(* Logix 5000 project; controller test vendor 1 type 14 code 151 rev 32.13; software revision 32.02; part 2 of 4 *)

        [600].Status := 2, [601].Status := 2, [602].Status := 2, [603].Status := 2, [604].Status := 2, [605].Status := 2, [606].Status := 2, [607].Status := 2, [608].Status := 2, [609].Status := 2, [610].Status := 2, [611].Status := 2, [612].Status := 2, [613].Status := 2, [614].Status := 2, [615].Status := 2, [616].Status := 2, [617].Status := 2, [618].Status := 2, [619].Status := 2, [620].Status := 2, [621].Status := 2, [622].Status := 2, [623].Status := 2, [624].Status := 2, [625].Status := 2, [626].Status := 2, [627].Status := 2, [628].Status := 2, [629].Status := 2, [630].Status := 2, [631].Status := 2, [632].Status := 2, [633].Status := 2, [634].Status := 2, [635].Status := 2, [636].Status := 2, [637].Status := 2, [638].Status := 2, [639].Status := 2, [640].Status := 2, [641].Status := 2, [642].Status := 2, [643].Status := 2, [644].Status := 2, [645].Status := 2, [646].Status := 2, [647].Status := 2, [648].Status := 2, [649].Status := 2, [650].Status := 2, [651].Status := 2, [652].Status := 2, [653].Status := 2, [654].Status := 2, [655].Status := 2, [656].Status := 2, [657].Status := 2, [658].Status := 2, [659].Status := 2,
        [660].Status := 2, [661].Status := 2, [662].Status := 2, [663].Status := 2, [664].Status := 2, [665].Status := 2, [666].Status := 2, [667].Status := 2, [668].Status := 2, [669].Status := 2, [670].Status := 2, [671].Status := 2, [672].Status := 2, [673].Status := 2, [674].Status := 2, [675].Status := 2, [676].Status := 2, [677].Status := 2, [678].Status := 2, [679].Status := 2, [680].Status := 2, [681].Status := 2, [682].Status := 2, [683].Status := 2, [684].Status := 2, [685].Status := 2, [686].Status := 2, [687].Status := 2, [688].Status := 2, [689].Status := 2, [690].Status := 2, [691].Status := 2, [692].Status := 2, [693].Status := 2, [694].Status := 2, [695].Status := 2, [696].Status := 2, [697].Status := 2, [698].Status := 2, [699].Status := 2, [700].Status := 2, [701].Status := 2, [702].Status := 2, [703].Status := 2, [704].Status := 2, [705].Status := 2, [706].Status := 2, [707].Status := 2, [708].Status := 2, [709].Status := 2, [710].Status := 2, [711].Status := 2, [712].Status := 2, [713].Status := 2, [714].Status := 2, [715].Status := 2, [716].Status := 2, [717].Status := 2, [718].Status := 2, [719].Status := 2,
        [720].Status := 2, [721].Status := 2, [722].Status := 2, [723].Status := 2, [724].Status := 2, [725].Status := 2, [726].Status := 2, [727].Status := 2, [728].Status := 2, [729].Status := 2, [730].Status := 2, [731].Status := 2, [732].Status := 2, [733].Status := 2, [734].Status := 2, [735].Status := 2, [736].Status := 2, [737].Status := 2, [738].Status := 2, [739].Status := 2, [740].Status := 2, [741].Status := 2, [742].Status := 2, [743].Status := 2, [744].Status := 2, [745].Status := 2, [746].Status := 2, [747].Status := 2, [748].Status := 2, [749].Status := 2, [750].Status := 2, [751].Status := 2, [752].Status := 2, [753].Status := 2, [754].Status := 2, [755].Status := 2, [756].Status := 2, [757].Status := 2, [758].Status := 2, [759].Status := 2, [760].Status := 2, [761].Status := 2, [762].Status := 2, [763].Status := 2, [764].Status := 2, [765].Status := 2, [766].Status := 2, [767].Status := 2, [768].Status := 2, [769].Status := 2, [770].Status := 2, [771].Status := 2, [772].Status := 2, [773].Status := 2, [774].Status := 2, [775].Status := 2, [776].Status := 2, [777].Status := 2, [778].Status := 2, [779].Status := 2,
        [780].Status := 2, [781].Status := 2, [782].Status := 2, [783].Status := 2, [784].Status := 2, [785].Status := 2, [786].Status := 2, [787].Status := 2, [788].Status := 2, [789].Status := 2, [790].Status := 2, [791].Status := 2, [792].Status := 2, [793].Status := 2, [794].Status := 2, [795].Status := 2, [796].Status := 2, [797].Status := 2, [798].Status := 2, [799].Status := 2, [800].Status := 2, [801].Status := 2, [802].Status := 2, [803].Status := 2, [804].Status := 2, [805].Status := 2, [806].Status := 2, [807].Status := 2, [808].Status := 2, [809].Status := 2, [810].Status := 2, [811].Status := 2, [812].Status := 2, [813].Status := 2, [814].Status := 2, [815].Status := 2, [816].Status := 2, [817].Status := 2, [818].Status := 2, [819].Status := 2, [820].Status := 2, [821].Status := 2, [822].Status := 2, [823].Status := 2, [824].Status := 2, [825].Status := 2, [826].Status := 2, [827].Status := 2, [828].Status := 2, [829].Status := 2, [830].Status := 2, [831].Status := 2, [832].Status := 2, [833].Status := 2, [834].Status := 2, [835].Status := 2, [836].Status := 2, [837].Status := 2, [838].Status := 2, [839].Status := 2,
        [840].Status := 2, [841].Status := 2, [842].Status := 2, [843].Status := 2, [844].Status := 2, [845].Status := 2, [846].Status := 2, [847].Status := 2, [848].Status := 2, [849].Status := 2, [850].Status := 2, [851].Status := 2, [852].Status := 2, [853].Status := 2, [854].Status := 2, [855].Status := 2, [856].Status := 2, [857].Status := 2, [858].Status := 2, [859].Status := 2, [860].Status := 2, [861].Status := 2, [862].Status := 2, [863].Status := 2, [864].Status := 2, [865].Status := 2, [866].Status := 2, [867].Status := 2, [868].Status := 2, [869].Status := 2, [870].Status := 2, [871].Status := 2, [872].Status := 2, [873].Status := 2, [874].Status := 2, [875].Status := 2, [876].Status := 2, [877].Status := 2, [878].Status := 2, [879].Status := 2, [880].Status := 2, [881].Status := 2, [882].Status := 2, [883].Status := 2, [884].Status := 2, [885].Status := 2, [886].Status := 2, [887].Status := 2, [888].Status := 2, [889].Status := 2, [890].Status := 2, [891].Status := 2, [892].Status := 2, [893].Status := 2, [894].Status := 2, [895].Status := 2, [896].Status := 2, [897].Status := 2, [898].Status := 2, [899].Status := 2,
        [900].Status := 2, [901].Status := 2, [902].Status := 2, [903].Status := 2, [904].Status := 2, [905].Status := 2, [906].Status := 2, [907].Status := 2, [908].Status := 2, [909].Status := 2, [910].Status := 2, [911].Status := 2, [912].Status := 2, [913].Status := 2, [914].Status := 2, [915].Status := 2, [916].Status := 2, [917].Status := 2, [918].Status := 2, [919].Status := 2, [920].Status := 2, [921].Status := 2, [922].Status := 2, [923].Status := 2, [924].Status := 2, [925].Status := 2, [926].Status := 2, [927].Status := 2, [928].Status := 2, [929].Status := 2, [930].Status := 2, [931].Status := 2, [932].Status := 2, [933].Status := 2, [934].Status := 2, [935].Status := 2, [936].Status := 2, [937].Status := 2, [938].Status := 2, [939].Status := 2, [940].Status := 2, [941].Status := 2, [942].Status := 2, [943].Status := 2, [944].Status := 2, [945].Status := 2, [946].Status := 2, [947].Status := 2, [948].Status := 2, [949].Status := 2, [950].Status := 2, [951].Status := 2, [952].Status := 2, [953].Status := 2, [954].Status := 2, [955].Status := 2, [956].Status := 2, [957].Status := 2, [958].Status := 2, [959].Status := 2,
        [960].Status := 2, [961].Status := 2, [962].Status := 2, [963].Status := 2, [964].Status := 2, [965].Status := 2, [966].Status := 2, [967].Status := 2, [968].Status := 2, [969].Status := 2, [970].Status := 2, [971].Status := 2, [972].Status := 2, [973].Status := 2, [974].Status := 2, [975].Status := 2, [976].Status := 2, [977].Status := 2, [978].Status := 2, [979].Status := 2, [980].Status := 2, [981].Status := 2, [982].Status := 2, [983].Status := 2, [984].Status := 2, [985].Status := 2, [986].Status := 2, [987].Status := 2, [988].Status := 2, [989].Status := 2, [990].Status := 2, [991].Status := 2, [992].Status := 2, [993].Status := 2, [994].Status := 2, [995].Status := 2, [996].Status := 2, [997].Status := 2, [998].Status := 2, [999].Status := 2, [1000].Status := 2, [1001].Status := 2, [1002].Status := 2);
   AlarmPressureHigh : REAL;
   AnalogFlowAirHAlarm : ALIAS FOR Local:2:I.Ch1HAlarm;
   AnalogFlowAirLAlarm : ALIAS FOR Local:2:I.Ch1LAlarm;
   AnalogFlowO2HAlarm : ALIAS FOR Local:2:I.Ch0HAlarm;
   AnalogFlowO2LAlarm : ALIAS FOR Local:2:I.Ch0LAlarm;
   AnalogInputFlow : ALIAS FOR Local:2:I.Ch3Data;
   AnalogInputFlowAir : ALIAS FOR Local:2:I.Ch1Data;
   AnalogInputFlowO2 : ALIAS FOR Local:2:I.Ch0Data;
   AnalogInputPressure : ALIAS FOR Local:2:I.Ch2Data;
   AnalogOutFlowAir : ALIAS FOR Local:2:O.Ch1Data;
   AnalogOutFlowO2 : ALIAS FOR Local:2:O.Ch0Data;
   AnalogPressureHAlarm : ALIAS FOR Local:2:I.Ch2HAlarm;
   AnalogPressureLAlarm : ALIAS FOR Local:2:I.Ch2LAlarm;
   ARRAYSHIFT : AOI_ARRAYSHIFT;
   avgCrsDyn : REAL := 0.44807863;   // 1 min avg of dynamic respiratory system compliance in ml/cmH2O, from measAvgCalc()
   avgCrsQStat : REAL := 0.50136733;   // 1 min avg of quasistatic respiratory system compliance in ml/cmH2O, from measAvgCalc()
   avgFlowImax : REAL := 18987.0;   // 1 min avg of max insp flow in l/min, from measAvgCalc()
   avgMV : REAL := 41214.273;   // 1 min avg of minute ventilation in l/min, from measAvgCalc()
   avgPEEP : REAL := 4402.0;   // 1 min avg of positive end expiratory pressure in cmH2O, from measAvgCalc()
   avgPpeak : REAL := 10534.0;   // 1 min avg of peak insp pressure in cmH2O, from measAvgCalc()
   avgPplat : REAL := 9882.25;   // 1 min avg of plateau insp pressure in cmH2O, from measAvgCalc()
   avgRaw : REAL := 2.059567;   // 1 min avg of airway resistance in cmH2O/l/s, from measAvgCalc()
   avgRR : REAL := 15.0;   // 1 min avg of respiratory rate in 1/min, from measAvgCalc()
   avgVti : REAL := 2747.6182;   // 1 min avg of insp tidal volume in ml, from measAvgCalc()
   BackingTag : MOTION_INSTRUCTION := (FLAGS := 33554432);
   BreathDetect : BOOL;
   BreathDuration : INT := 4;
   BreathDurationArr : REAL[50] := ([0] := -1.0, [1] := -1.0, [2] := -1.0, [3] := -1.0, [4] := -1.0, [5] := -1.0, [6] := -1.0, [7] := -1.0, [8] := -1.0, [9] := -1.0, [10] := -1.0, [11] := -1.0, [12] := -1.0, [13] := -1.0, [14] := -1.0, [15] := -1.0, [16] := -1.0, [17] := -1.0, [18] := -1.0, [19] := -1.0, [20] := -1.0, [21] := -1.0, [22] := -1.0, [23] := -1.0, [24] := -1.0, [25] := -1.0, [26] := -1.0, [27] := -1.0, [28] := -1.0, [29] := -1.0, [30] := -1.0, [31] := -1.0, [32] := -1.0, [33] := -1.0, [34] := -1.0, [35] := -1.0, [36] := -1.0, [37] := -1.0, [38] := -1.0, [39] := -1.0, [40] := -1.0, [41] := -1.0, [42] := -1.0, [43] := -1.0, [44] := -1.0, [45] := -1.0, [46] := -1.0, [47] := -1.0, [48] := -1.0, [49] := -1.0);   // 50 length array with seconds for each breath for calculation of minute avgVentStateArr. Calcualted from knowing meas at 100Hz for all breath data
   BreathDurationInMS : REAL := 4000.0002;
   CalcMe : BOOL;
   CalcNewData : BOOL;
   ConstansFlowNrCalc : REAL := 40.0;
   ConstantFlowNrOfAdjustments : REAL := 40.0;
   ConstantFlowTimeInMS : REAL := 400.0;
   ConstantInspiratoryFlow : REAL := 72.0;
   counter : DINT := 787;   // Counter for Flow fill array
   CrsDyn : REAL := 0.5221349;   // dynamic respiraotry system compliance in ml/cmH2O
   CrsDynArr : REAL[50];   // 50 length array with dynamic respiraotry system compliance in ml/cmH2O, from measCalc()
   CrsQStat : REAL := 0.59738743;   // quasistatic respiratory system compliance in ml/cmH2O
   CrsQStatArr : REAL[50];   // 50 length array with quasistatic respiratory system compliance in ml/cmH2O, from measCalc()
   CsumData : DINT := 659;
   CsumDataOld : DINT := 659;
   data_changed : BOOL;
   DymmyMaster : AXIS_VIRTUAL;
   DymmySlave : AXIS_VIRTUAL;
   endI : DINT;
   EndPoint : INT := 194;
   Exp : BOOL;
   expCount : INT;   // between 1-1000 to indicate where valveCtrl should read from expOpenCloseCtrl[]
   expCountLength : INT := 300;   // between 1-1000 to indicate when valveCtrl should stop reading from expOpenCloseCtrl[], copied from nextExpCountLength by ISR_ValveCtrl()
   expCountlengthCalc : REAL := 300.00003;
   expCountLengthNew : REAL := 300.0;
   expEndI : INT;
   expOpen : ALIAS FOR Local:1:O.Data.0;
   expOpenCloseCtrl : INT[1000] := ([0] := 1, [1] := 1, [2] := 1, [3] := 1, [4] := 1, [5] := 1, [6] := 1, [7] := 1, [8] := 1, [9] := 1, [10] := 1, [11] := 1, [12] := 1, [13] := 1, [14] := 1, [15] := 1, [16] := 1, [17] := 1, [18] := 1, [19] := 1, [20] := 1, [21] := 1, [22] := 1, [23] := 1, [24] := 1, [25] := 1, [26] := 1, [27] := 1, [28] := 1, [29] := 1, [30] := 1, [31] := 1, [32] := 1, [33] := 1, [34] := 1, [35] := 1, [36] := 1, [37] := 1, [38] := 1, [39] := 1, [40] := 1, [41] := 1, [42] := 1, [43] := 1, [44] := 1, [45] := 1, [46] := 1, [47] := 1, [48] := 1, [49] := 1, [50] := 1, [51] := 1, [52] := 1, [53] := 1, [54] := 1, [55] := 1, [56] := 1, [57] := 1, [58] := 1, [59] := 1,
        [60] := 1, [61] := 1, [62] := 1, [63] := 1, [64] := 1, [65] := 1, [66] := 1, [67] := 1, [68] := 1, [69] := 1, [70] := 1, [71] := 1, [72] := 1, [73] := 1, [74] := 1, [75] := 1, [76] := 1, [77] := 1, [78] := 1, [79] := 1, [80] := 1, [81] := 1, [82] := 1, [83] := 1, [84] := 1, [85] := 1, [86] := 1, [87] := 1, [88] := 1, [89] := 1, [90] := 1, [91] := 1, [92] := 1, [93] := 1, [94] := 1, [95] := 1, [96] := 1, [97] := 1, [98] := 1, [99] := 1, [100] := 1, [101] := 1, [102] := 1, [103] := 1, [104] := 1, [105] := 1, [106] := 1, [107] := 1, [108] := 1, [109] := 1, [110] := 1, [111] := 1, [112] := 1, [113] := 1, [114] := 1, [115] := 1, [116] := 1, [117] := 1, [118] := 1, [119] := 1,
        [120] := 1, [121] := 1, [122] := 1, [123] := 1, [124] := 1, [125] := 1, [126] := 1, [127] := 1, [128] := 1, [129] := 1, [130] := 1, [131] := 1, [132] := 1, [133] := 1, [134] := 1, [135] := 1, [136] := 1, [137] := 1, [138] := 1, [139] := 1, [140] := 1, [141] := 1, [142] := 1, [143] := 1, [144] := 1, [145] := 1, [146] := 1, [147] := 1, [148] := 1, [149] := 1, [150] := 1, [151] := 1, [152] := 1, [153] := 1, [154] := 1, [155] := 1, [156] := 1, [157] := 1, [158] := 1, [159] := 1, [160] := 1, [161] := 1, [162] := 1, [163] := 1, [164] := 1, [165] := 1, [166] := 1, [167] := 1, [168] := 1, [169] := 1, [170] := 1, [171] := 1, [172] := 1, [173] := 1, [174] := 1, [175] := 1, [176] := 1, [177] := 1, [178] := 1, [179] := 1,
        [180] := 1, [181] := 1, [182] := 1, [183] := 1, [184] := 1, [185] := 1, [186] := 1, [187] := 1, [188] := 1, [189] := 1, [190] := 1, [191] := 1, [192] := 1, [193] := 1, [194] := 1, [195] := 1, [196] := 1, [197] := 1, [198] := 1, [199] := 1, [200] := 1, [201] := 1, [202] := 1, [203] := 1, [204] := 1, [205] := 1, [206] := 1, [207] := 1, [208] := 1, [209] := 1, [210] := 1, [211] := 1, [212] := 1, [213] := 1, [214] := 1, [215] := 1, [216] := 1, [217] := 1, [218] := 1, [219] := 1, [220] := 1, [221] := 1, [222] := 1, [223] := 1, [224] := 1, [225] := 1, [226] := 1, [227] := 1, [228] := 1, [229] := 1, [230] := 1, [231] := 1, [232] := 1, [233] := 1, [234] := 1, [235] := 1, [236] := 1, [237] := 1, [238] := 1, [239] := 1,
        [240] := 1, [241] := 1, [242] := 1, [243] := 1, [244] := 1, [245] := 1, [246] := 1, [247] := 1, [248] := 1, [249] := 1, [250] := 1, [251] := 1, [252] := 1, [253] := 1, [254] := 1, [255] := 1, [256] := 1, [257] := 1, [258] := 1, [259] := 1, [260] := 1, [261] := 1, [262] := 1, [263] := 1, [264] := 1, [265] := 1, [266] := 1, [267] := 1, [268] := 1, [269] := 1, [270] := 1, [271] := 1, [272] := 1, [273] := 1, [274] := 1, [275] := 1, [276] := 1, [277] := 1, [278] := 1, [279] := 1, [280] := 1, [281] := 1, [282] := 1, [283] := 1, [284] := 1, [285] := 1, [286] := 1, [287] := 1, [288] := 1, [289] := 1, [290] := 1, [291] := 1, [292] := 1, [293] := 1, [294] := 1, [295] := 1, [296] := 1, [297] := 1, [298] := 1, [299] := 1);   // 1000 length array with open (1) or close (0) for exp valve, moved from nextexpOpenCloseCtrl[] by ISR_ValveCtrl()
   expOpenCloseCtrlNew : INT[1000] := ([0] := 1, [1] := 1, [2] := 1, [3] := 1, [4] := 1, [5] := 1, [6] := 1, [7] := 1, [8] := 1, [9] := 1, [10] := 1, [11] := 1, [12] := 1, [13] := 1, [14] := 1, [15] := 1, [16] := 1, [17] := 1, [18] := 1, [19] := 1, [20] := 1, [21] := 1, [22] := 1, [23] := 1, [24] := 1, [25] := 1, [26] := 1, [27] := 1, [28] := 1, [29] := 1, [30] := 1, [31] := 1, [32] := 1, [33] := 1, [34] := 1, [35] := 1, [36] := 1, [37] := 1, [38] := 1, [39] := 1, [40] := 1, [41] := 1, [42] := 1, [43] := 1, [44] := 1, [45] := 1, [46] := 1, [47] := 1, [48] := 1, [49] := 1, [50] := 1, [51] := 1, [52] := 1, [53] := 1, [54] := 1, [55] := 1, [56] := 1, [57] := 1, [58] := 1, [59] := 1,
        [60] := 1, [61] := 1, [62] := 1, [63] := 1, [64] := 1, [65] := 1, [66] := 1, [67] := 1, [68] := 1, [69] := 1, [70] := 1, [71] := 1, [72] := 1, [73] := 1, [74] := 1, [75] := 1, [76] := 1, [77] := 1, [78] := 1, [79] := 1, [80] := 1, [81] := 1, [82] := 1, [83] := 1, [84] := 1, [85] := 1, [86] := 1, [87] := 1, [88] := 1, [89] := 1, [90] := 1, [91] := 1, [92] := 1, [93] := 1, [94] := 1, [95] := 1, [96] := 1, [97] := 1, [98] := 1, [99] := 1, [100] := 1, [101] := 1, [102] := 1, [103] := 1, [104] := 1, [105] := 1, [106] := 1, [107] := 1, [108] := 1, [109] := 1, [110] := 1, [111] := 1, [112] := 1, [113] := 1, [114] := 1, [115] := 1, [116] := 1, [117] := 1, [118] := 1, [119] := 1,
        [120] := 1, [121] := 1, [122] := 1, [123] := 1, [124] := 1, [125] := 1, [126] := 1, [127] := 1, [128] := 1, [129] := 1, [130] := 1, [131] := 1, [132] := 1, [133] := 1, [134] := 1, [135] := 1, [136] := 1, [137] := 1, [138] := 1, [139] := 1, [140] := 1, [141] := 1, [142] := 1, [143] := 1, [144] := 1, [145] := 1, [146] := 1, [147] := 1, [148] := 1, [149] := 1, [150] := 1, [151] := 1, [152] := 1, [153] := 1, [154] := 1, [155] := 1, [156] := 1, [157] := 1, [158] := 1, [159] := 1, [160] := 1, [161] := 1, [162] := 1, [163] := 1, [164] := 1, [165] := 1, [166] := 1, [167] := 1, [168] := 1, [169] := 1, [170] := 1, [171] := 1, [172] := 1, [173] := 1, [174] := 1, [175] := 1, [176] := 1, [177] := 1, [178] := 1, [179] := 1,
        [180] := 1, [181] := 1, [182] := 1, [183] := 1, [184] := 1, [185] := 1, [186] := 1, [187] := 1, [188] := 1, [189] := 1, [190] := 1, [191] := 1, [192] := 1, [193] := 1, [194] := 1, [195] := 1, [196] := 1, [197] := 1, [198] := 1, [199] := 1, [200] := 1, [201] := 1, [202] := 1, [203] := 1, [204] := 1, [205] := 1, [206] := 1, [207] := 1, [208] := 1, [209] := 1, [210] := 1, [211] := 1, [212] := 1, [213] := 1, [214] := 1, [215] := 1, [216] := 1, [217] := 1, [218] := 1, [219] := 1, [220] := 1, [221] := 1, [222] := 1, [223] := 1, [224] := 1, [225] := 1, [226] := 1, [227] := 1, [228] := 1, [229] := 1, [230] := 1, [231] := 1, [232] := 1, [233] := 1, [234] := 1, [235] := 1, [236] := 1, [237] := 1, [238] := 1, [239] := 1,
        [240] := 1, [241] := 1, [242] := 1, [243] := 1, [244] := 1, [245] := 1, [246] := 1, [247] := 1, [248] := 1, [249] := 1, [250] := 1, [251] := 1, [252] := 1, [253] := 1, [254] := 1, [255] := 1, [256] := 1, [257] := 1, [258] := 1, [259] := 1, [260] := 1, [261] := 1, [262] := 1, [263] := 1, [264] := 1, [265] := 1, [266] := 1, [267] := 1, [268] := 1, [269] := 1, [270] := 1, [271] := 1, [272] := 1, [273] := 1, [274] := 1, [275] := 1, [276] := 1, [277] := 1, [278] := 1, [279] := 1, [280] := 1, [281] := 1, [282] := 1, [283] := 1, [284] := 1, [285] := 1, [286] := 1, [287] := 1, [288] := 1, [289] := 1, [290] := 1, [291] := 1, [292] := 1, [293] := 1, [294] := 1, [295] := 1, [296] := 1, [297] := 1, [298] := 1, [299] := 1);
   expStartI : INT;
   expTimeInMS : REAL := 3000.0002;
   F1_pushed_new : BOOL;
   F1_pushed_old : BOOL;
   F2_pushed_new : BOOL;
   F2_pushed_old : BOOL;
   F3_pushed_new : BOOL;
   F3_pushed_old : BOOL;
   FFL_ctr : CONTROL := (LEN := 2000, POS := 691);
   Fill : AOI_FillArrayReal := (Len := 650);
   Fill50 : AOI_FillArrayReal50 := (Source := -1, Len := 50);
   Fillint : AOI_FillArrayInt := (Source := 1, Len := 300);
   FillLoop : AOI_FillArray_Real2D := (Len := 2000);
   FiO2 : INT := 25;   // 25-100%
   FiO2Running : INT := 25;
   Floor : AOI_Floor := (In_X := 40.000004);
   FlowAir : REAL[1000,2] := ([0,0] := 73.65, [1,0] := 73.65, [2,0] := 73.65, [3,0] := 73.65, [4,0] := 73.65, [5,0] := 73.65, [6,0] := 73.65, [7,0] := 73.65, [8,0] := 73.65, [9,0] := 73.65, [10,0] := 73.725, [11,0] := 73.725, [12,0] := 73.65, [13,0] := 73.65, [14,0] := 73.65, [15,0] := 73.65, [16,0] := 73.65, [17,0] := 73.725, [18,0] := 73.725, [19,0] := 73.725, [20,0] := 73.725, [21,0] := 73.725, [22,0] := 73.65, [23,0] := 73.65, [24,0] := 73.65, [25,0] := 73.65, [26,0] := 73.65, [27,0] := 73.65, [28,0] := 73.65, [29,0] := 73.65, [30,0] := 73.65, [31,0] := 73.65, [32,0] := 73.65, [33,0] := 73.65, [34,0] := 73.65, [35,0] := 73.65, [36,0] := 73.65, [37,0] := 73.65, [38,0] := 73.65, [39,0] := 73.65, [40,0] := 73.65, [41,0] := 73.725, [42,0] := 73.725, [43,0] := 73.725, [44,0] := 73.725, [45,0] := 73.725, [46,0] := 73.65, [47,0] := 73.65, [48,0] := 73.725, [49,0] := 73.725, [50,0] := 73.725, [51,0] := 73.65, [52,0] := 73.65, [53,0] := 73.65, [54,0] := 73.65, [55,0] := 73.65, [56,0] := 73.65, [57,0] := 73.65, [58,0] := 73.65, [59,0] := 73.65,
        [60,0] := 73.65, [61,0] := 73.65, [62,0] := 73.65, [63,0] := 73.65, [64,0] := 73.65, [65,0] := 73.65, [66,0] := 73.65, [67,0] := 73.65, [68,0] := 73.65, [69,0] := 73.65, [70,0] := 73.65, [71,0] := 73.65, [72,0] := 73.725, [73,0] := 73.725, [74,0] := 73.725, [75,0] := 73.65, [76,0] := 73.65, [77,0] := 73.65, [78,0] := 73.65, [79,0] := 73.65, [80,0] := 73.725, [81,0] := 73.725, [82,0] := 73.725, [83,0] := 73.725, [84,0] := 73.65, [85,0] := 73.65, [86,0] := 73.65, [87,0] := 73.65, [88,0] := 73.65, [89,0] := 73.65, [90,0] := 73.65, [91,0] := 73.65, [92,0] := 73.65, [93,0] := 73.65, [94,0] := 73.65, [95,0] := 73.65, [96,0] := 73.65, [97,0] := 73.65, [98,0] := 73.65, [99,0] := 73.65, [100,0] := 73.65, [101,0] := 73.65, [102,0] := 73.65, [103,0] := 73.65, [104,0] := 73.65, [105,0] := 73.65, [106,0] := 73.65, [107,0] := 73.65, [108,0] := 73.65, [109,0] := 73.65, [110,0] := 73.65, [111,0] := 73.725, [112,0] := 73.725, [113,0] := 73.725, [114,0] := 73.725, [115,0] := 73.725, [116,0] := 73.65, [117,0] := 73.65, [118,0] := 73.725, [119,0] := 73.725,
        [120,0] := 73.65, [121,0] := 73.65, [122,0] := 73.65, [123,0] := 73.65, [124,0] := 73.65, [125,0] := 73.65, [126,0] := 73.65, [127,0] := 73.65, [128,0] := 73.65, [129,0] := 73.65, [130,0] := 73.65, [131,0] := 73.65, [132,0] := 73.65, [133,0] := 73.65, [134,0] := 73.65, [135,0] := 73.65, [136,0] := 73.65, [137,0] := 73.65, [138,0] := 73.65, [139,0] := 73.65, [140,0] := 73.65, [141,0] := 73.65, [142,0] := 73.725, [143,0] := 73.725, [144,0] := 73.725, [145,0] := 73.725, [146,0] := 73.725, [147,0] := 73.65, [148,0] := 73.65, [149,0] := 73.725, [150,0] := 73.725, [151,0] := 73.725, [152,0] := 73.65, [153,0] := 73.65, [154,0] := 73.65, [155,0] := 73.65, [156,0] := 73.65, [157,0] := 73.65, [158,0] := 73.65, [159,0] := 73.65, [160,0] := 73.65, [161,0] := 73.65, [162,0] := 73.65, [163,0] := 73.65, [164,0] := 73.65, [165,0] := 73.65, [166,0] := 73.65, [167,0] := 73.65, [168,0] := 73.65, [169,0] := 73.65, [170,0] := 73.65, [171,0] := 73.65, [172,0] := 73.65, [173,0] := 73.725, [174,0] := 73.725, [175,0] := 73.725, [176,0] := 73.725, [177,0] := 73.725, [178,0] := 73.65, [179,0] := 73.65,
        [180,0] := 73.65, [181,0] := 73.725, [182,0] := 73.725, [183,0] := 73.65, [184,0] := 73.65, [185,0] := 73.65, [186,0] := 73.65, [187,0] := 73.65, [188,0] := 73.65, [189,0] := 73.65, [190,0] := 73.65, [191,0] := 73.65, [192,0] := 73.65, [193,0] := 73.65, [194,0] := 73.65, [195,0] := 73.65, [196,0] := 73.65, [197,0] := 73.65, [198,0] := 73.65, [199,0] := 73.65, [200,0] := 73.65, [201,0] := 73.65, [202,0] := 73.65, [203,0] := 73.65, [204,0] := 73.65, [205,0] := 73.725, [206,0] := 73.725, [207,0] := 73.65, [208,0] := 73.65, [209,0] := 73.65, [210,0] := 73.65, [211,0] := 73.65, [212,0] := 73.725, [213,0] := 73.725, [214,0] := 73.65, [215,0] := 73.65, [216,0] := 73.65, [217,0] := 73.65, [218,0] := 73.65, [219,0] := 73.65, [220,0] := 73.65, [221,0] := 73.65, [222,0] := 73.65, [223,0] := 73.65, [224,0] := 73.65, [225,0] := 73.65, [226,0] := 73.65, [227,0] := 73.65, [228,0] := 73.65, [229,0] := 73.65, [230,0] := 73.65, [231,0] := 73.65, [232,0] := 73.65, [233,0] := 73.65, [234,0] := 73.65, [235,0] := 73.65, [236,0] := 73.65, [237,0] := 73.65, [238,0] := 73.65, [239,0] := 73.65,
        [240,0] := 73.65, [241,0] := 73.65, [242,0] := 73.65, [243,0] := 73.725, [244,0] := 73.725, [245,0] := 73.725, [246,0] := 73.725, [247,0] := 73.725, [248,0] := 73.65, [249,0] := 73.65, [250,0] := 73.65, [251,0] := 73.65, [252,0] := 73.65, [253,0] := 73.65, [254,0] := 73.65, [255,0] := 73.65, [256,0] := 73.65, [257,0] := 73.65, [258,0] := 73.65, [259,0] := 73.65, [260,0] := 73.65, [261,0] := 73.65, [262,0] := 73.65, [263,0] := 73.65, [264,0] := 73.65, [265,0] := 73.65, [266,0] := 73.65, [267,0] := 73.725, [268,0] := 73.725, [269,0] := 73.725, [270,0] := 73.65, [271,0] := 73.65, [272,0] := 73.65, [273,0] := 73.65, [274,0] := 73.725, [275,0] := 73.725, [276,0] := 73.725, [277,0] := 73.725, [278,0] := 73.725, [279,0] := 73.65, [280,0] := 73.65, [281,0] := 73.65, [282,0] := 73.65, [283,0] := 73.65, [284,0] := 73.65, [285,0] := 73.65, [286,0] := 73.65, [287,0] := 73.65, [288,0] := 73.65, [289,0] := 73.65, [290,0] := 73.65, [291,0] := 73.65, [292,0] := 73.65, [293,0] := 73.65, [294,0] := 73.65, [295,0] := 73.65, [296,0] := 73.65, [297,0] := 73.65, [298,0] := 73.65, [299,0] := 73.725,
        [300,0] := 73.725, [301,0] := 73.725, [302,0] := 73.725, [303,0] := 73.65, [304,0] := 73.65, [305,0] := 73.65, [306,0] := 73.65, [307,0] := 73.65, [308,0] := 73.65, [309,0] := 73.65, [310,0] := 73.65, [311,0] := 73.65, [312,0] := 73.65, [313,0] := 73.65, [314,0] := 73.65, [315,0] := 73.65, [316,0] := 73.65, [317,0] := 73.65, [318,0] := 73.65, [319,0] := 73.65, [320,0] := 73.65, [321,0] := 73.65, [322,0] := 73.65, [323,0] := 73.65, [324,0] := 73.65, [325,0] := 73.65, [326,0] := 73.65, [327,0] := 73.65, [328,0] := 73.65, [329,0] := 73.65, [330,0] := 73.725, [331,0] := 73.725, [332,0] := 73.725, [333,0] := 73.725, [334,0] := 73.725, [335,0] := 73.65, [336,0] := 73.65, [337,0] := 73.725, [338,0] := 73.725, [339,0] := 73.725, [340,0] := 73.725, [341,0] := 73.725, [342,0] := 73.65, [343,0] := 73.65, [344,0] := 73.65, [345,0] := 73.65, [346,0] := 73.65, [347,0] := 73.65, [348,0] := 73.65, [349,0] := 73.65, [350,0] := 73.65, [351,0] := 73.65, [352,0] := 73.65, [353,0] := 73.65, [354,0] := 73.65, [355,0] := 73.65, [356,0] := 73.65, [357,0] := 73.65, [358,0] := 73.65, [359,0] := 73.65,
        [360,0] := 73.65, [361,0] := 73.725, [362,0] := 73.725, [363,0] := 73.725, [364,0] := 73.725, [365,0] := 73.725, [366,0] := 73.65, [367,0] := 73.65, [368,0] := 73.65, [369,0] := 73.65, [370,0] := 73.65, [371,0] := 73.65, [372,0] := 73.65, [373,0] := 73.65, [374,0] := 73.65, [375,0] := 73.65, [376,0] := 73.65, [377,0] := 73.65, [378,0] := 73.65, [379,0] := 73.65, [380,0] := 73.65, [381,0] := 73.65, [382,0] := 73.65, [383,0] := 73.65, [384,0] := 73.65, [385,0] := 73.65, [386,0] := 73.65, [387,0] := 73.65, [388,0] := 73.65, [389,0] := 73.65, [390,0] := 73.65, [391,0] := 73.65, [392,0] := 73.65, [393,0] := 73.725, [394,0] := 73.725, [395,0] := 73.725, [396,0] := 73.725, [397,0] := 73.65, [398,0] := 73.65, [399,0] := 73.65, [400,0] := 73.65, [401,0] := 73.65, [402,0] := 73.65, [403,0] := 73.65, [404,0] := 73.65, [405,0] := 73.65, [406,0] := 73.65, [407,0] := 73.65, [408,0] := 73.65, [409,0] := 73.65, [410,0] := 73.65, [411,0] := 73.65, [412,0] := 73.65, [413,0] := 73.65, [414,0] := 73.65, [415,0] := 73.65, [416,0] := 73.65, [417,0] := 73.65, [418,0] := 73.65, [419,0] := 73.65,
        [420,0] := 73.65, [421,0] := 73.65, [422,0] := 73.65, [423,0] := 73.65, [424,0] := 73.725, [425,0] := 73.725, [426,0] := 73.725, [427,0] := 73.725, [428,0] := 73.725, [429,0] := 73.65, [430,0] := 73.65, [431,0] := 73.725, [432,0] := 73.725, [433,0] := 73.65, [434,0] := 73.65, [435,0] := 73.65, [436,0] := 73.65, [437,0] := 73.65, [438,0] := 73.65, [439,0] := 73.65, [440,0] := 73.65, [441,0] := 73.65, [442,0] := 73.65, [443,0] := 73.65, [444,0] := 73.65, [445,0] := 73.65, [446,0] := 73.65, [447,0] := 73.65, [448,0] := 73.65, [449,0] := 73.65, [450,0] := 73.65, [451,0] := 73.65, [452,0] := 73.65, [453,0] := 73.65, [454,0] := 73.65, [455,0] := 73.65, [456,0] := 73.65, [457,0] := 73.65, [458,0] := 73.65, [459,0] := 73.65, [460,0] := 73.65, [461,0] := 73.65, [462,0] := 73.725, [463,0] := 73.725, [464,0] := 73.725, [465,0] := 73.725, [466,0] := 73.725, [467,0] := 73.65, [468,0] := 73.65, [469,0] := 73.65, [470,0] := 73.725, [471,0] := 73.725, [472,0] := 73.65, [473,0] := 73.65, [474,0] := 73.65, [475,0] := 73.65, [476,0] := 73.65, [477,0] := 73.65, [478,0] := 73.65, [479,0] := 73.65,
        [480,0] := 73.65, [481,0] := 73.65, [482,0] := 73.65, [483,0] := 73.65, [484,0] := 73.65, [485,0] := 73.65, [486,0] := 73.725, [487,0] := 73.725, [488,0] := 73.725, [489,0] := 73.65, [490,0] := 73.65, [491,0] := 73.65, [492,0] := 73.65, [493,0] := 73.65, [494,0] := 73.725, [495,0] := 73.725, [496,0] := 73.725, [497,0] := 73.725, [498,0] := 73.65, [499,0] := 73.65, [500,0] := 73.65, [501,0] := 73.725, [502,0] := 73.725, [503,0] := 73.65, [504,0] := 73.65, [505,0] := 73.65, [506,0] := 73.65, [507,0] := 73.65, [508,0] := 73.65, [509,0] := 73.65, [510,0] := 73.65, [511,0] := 73.65, [512,0] := 73.65, [513,0] := 73.65, [514,0] := 73.65, [515,0] := 73.65, [516,0] := 73.65, [517,0] := 73.65, [518,0] := 73.65, [519,0] := 73.65, [520,0] := 73.65, [521,0] := 73.65, [522,0] := 73.65, [523,0] := 73.65, [524,0] := 73.65, [525,0] := 73.725, [526,0] := 73.725, [527,0] := 73.65, [528,0] := 73.65, [529,0] := 73.65, [530,0] := 73.65, [531,0] := 73.65, [532,0] := 73.725, [533,0] := 73.725, [534,0] := 73.725, [535,0] := 73.725, [536,0] := 73.725, [537,0] := 73.65, [538,0] := 73.65, [539,0] := 73.65,
        [540,0] := 73.65, [541,0] := 73.65, [542,0] := 73.65, [543,0] := 73.65, [544,0] := 73.65, [545,0] := 73.65, [546,0] := 73.65, [547,0] := 73.65, [548,0] := 73.65, [549,0] := 73.65, [550,0] := 73.65, [551,0] := 73.65, [552,0] := 73.65, [553,0] := 73.65, [554,0] := 73.65, [555,0] := 73.65, [556,0] := 73.65, [557,0] := 73.65, [558,0] := 73.65, [559,0] := 73.65, [560,0] := 73.65, [561,0] := 73.65, [562,0] := 73.65, [563,0] := 73.725, [564,0] := 73.725, [565,0] := 73.725, [566,0] := 73.725, [567,0] := 73.725, [568,0] := 73.65, [569,0] := 73.65, [570,0] := 73.725, [571,0] := 73.725, [572,0] := 73.725, [573,0] := 73.725, [574,0] := 73.725, [575,0] := 73.65, [576,0] := 73.65, [577,0] := 73.65, [578,0] := 73.65, [579,0] := 73.65, [580,0] := 73.65, [581,0] := 73.65, [582,0] := 73.65, [583,0] := 73.65, [584,0] := 73.65, [585,0] := 73.65, [586,0] := 73.65, [587,0] := 73.65, [588,0] := 73.65, [589,0] := 73.65, [590,0] := 73.65, [591,0] := 73.65, [592,0] := 73.65, [593,0] := 73.65, [594,0] := 73.65, [595,0] := 73.65, [596,0] := 73.65, [597,0] := 73.65, [598,0] := 73.65, [599,0] := 73.65,
        [600,0] := 73.65, [601,0] := 73.65, [602,0] := 73.725, [603,0] := 73.725, [604,0] := 73.65, [605,0] := 73.65, [606,0] := 73.65, [607,0] := 73.65, [608,0] := 73.65, [609,0] := 73.65, [610,0] := 73.65, [611,0] := 73.65, [612,0] := 73.65, [613,0] := 73.65, [614,0] := 73.65, [615,0] := 73.65, [616,0] := 73.65, [617,0] := 73.65, [618,0] := 73.65, [619,0] := 73.65, [620,0] := 73.65, [621,0] := 73.65, [622,0] := 73.65, [623,0] := 73.65, [624,0] := 73.65, [625,0] := 73.65, [626,0] := 73.725, [627,0] := 73.725, [628,0] := 73.725, [629,0] := 73.725, [630,0] := 73.725, [631,0] := 73.65, [632,0] := 73.65, [633,0] := 73.65, [634,0] := 73.65, [635,0] := 73.65, [636,0] := 73.65, [637,0] := 73.65, [638,0] := 73.65, [639,0] := 73.65, [640,0] := 73.65, [641,0] := 73.65, [642,0] := 73.65, [643,0] := 73.65, [644,0] := 73.65, [645,0] := 73.65, [646,0] := 73.65, [647,0] := 73.65, [648,0] := 73.65, [649,0] := 73.65, [650,0] := 73.725, [651,0] := 73.725, [652,0] := 73.65, [653,0] := 73.65, [654,0] := 73.65, [655,0] := 73.65, [656,0] := 73.65, [657,0] := 73.725, [658,0] := 73.725, [659,0] := 73.725,
        [660,0] := 73.725, [661,0] := 73.725, [662,0] := 73.65, [663,0] := 73.65, [664,0] := 73.65, [665,0] := 73.65, [666,0] := 73.65, [667,0] := 73.65, [668,0] := 73.65, [669,0] := 73.65, [670,0] := 73.65, [671,0] := 73.65, [672,0] := 73.65, [673,0] := 73.65, [674,0] := 73.65, [675,0] := 73.65, [676,0] := 73.65, [677,0] := 73.65, [678,0] := 73.65, [679,0] := 73.65, [680,0] := 73.65, [681,0] := 73.65, [682,0] := 73.65, [683,0] := 73.65, [684,0] := 73.65, [685,0] := 73.65, [686,0] := 73.65, [687,0] := 73.65, [688,0] := 73.65, [689,0] := 73.725, [690,0] := 73.725, [691,0] := 73.725, [692,0] := 73.725, [693,0] := 73.65, [694,0] := 73.65, [695,0] := 73.65, [696,0] := 73.725, [697,0] := 73.725, [698,0] := 73.725, [699,0] := 73.725, [700,0] := 73.725, [701,0] := 73.65, [702,0] := 73.65, [703,0] := 73.65, [704,0] := 73.65, [705,0] := 73.65, [706,0] := 73.65, [707,0] := 73.65, [708,0] := 73.65, [709,0] := 73.65, [710,0] := 73.65, [711,0] := 73.65, [712,0] := 73.65, [713,0] := 73.65, [714,0] := 73.65, [715,0] := 73.65, [716,0] := 73.65, [717,0] := 73.65, [718,0] := 73.65, [719,0] := 73.65,
        [720,0] := 73.725, [721,0] := 73.725, [722,0] := 73.725, [723,0] := 73.725, [724,0] := 73.725, [725,0] := 73.65, [726,0] := 73.65, [727,0] := 73.725, [728,0] := 73.725, [729,0] := 73.725, [730,0] := 73.65, [731,0] := 73.65, [732,0] := 73.65, [733,0] := 73.65, [734,0] := 73.65, [735,0] := 73.65, [736,0] := 73.65, [737,0] := 73.65, [738,0] := 73.65, [739,0] := 73.65, [740,0] := 73.65, [741,0] := 73.65, [742,0] := 73.65, [743,0] := 73.65, [744,0] := 73.65, [745,0] := 73.65, [746,0] := 73.65, [747,0] := 73.65, [748,0] := 73.65, [749,0] := 73.65, [750,0] := 73.65, [751,0] := 73.725, [752,0] := 73.725, [753,0] := 73.725, [754,0] := 73.725, [755,0] := 73.725, [756,0] := 73.65, [757,0] := 73.65, [758,0] := 73.725, [759,0] := 73.725, [760,0] := 73.725, [761,0] := 73.65, [762,0] := 73.65, [763,0] := 73.65, [764,0] := 73.65, [765,0] := 73.65, [766,0] := 73.65, [767,0] := 73.65, [768,0] := 73.65, [769,0] := 73.65, [770,0] := 73.65, [771,0] := 73.65, [772,0] := 73.65, [773,0] := 73.65, [774,0] := 73.65, [775,0] := 73.65, [776,0] := 73.65, [777,0] := 73.65, [778,0] := 73.65, [779,0] := 73.65,
        [780,0] := 73.65, [781,0] := 73.65, [782,0] := 73.725, [783,0] := 73.725, [784,0] := 73.725, [785,0] := 73.725, [786,0] := 73.725, [787,0] := 73.65, [788,0] := 73.65, [789,0] := 73.65, [790,0] := 73.725, [791,0] := 73.725, [792,0] := 73.65, [793,0] := 73.65, [794,0] := 73.65, [795,0] := 73.65, [796,0] := 73.65, [797,0] := 73.65, [798,0] := 73.65, [799,0] := 73.65, [800,0] := 73.65, [801,0] := 73.65, [802,0] := 73.65, [803,0] := 73.65, [804,0] := 73.65, [805,0] := 73.65, [806,0] := 73.65, [807,0] := 73.65, [808,0] := 73.65, [809,0] := 73.65, [810,0] := 73.65, [811,0] := 73.65, [812,0] := 73.65, [813,0] := 73.65, [814,0] := 73.725, [815,0] := 73.725, [816,0] := 73.725, [817,0] := 73.725, [818,0] := 73.725, [819,0] := 73.65, [820,0] := 73.65, [821,0] := 73.725, [822,0] := 73.725, [823,0] := 73.65, [824,0] := 73.65, [825,0] := 73.65, [826,0] := 73.65, [827,0] := 73.65, [828,0] := 73.65, [829,0] := 73.65, [830,0] := 73.65, [831,0] := 73.65, [832,0] := 73.65, [833,0] := 73.65, [834,0] := 73.65, [835,0] := 73.65, [836,0] := 73.65, [837,0] := 73.65, [838,0] := 73.65, [839,0] := 73.65,
        [840,0] := 73.65, [841,0] := 73.65, [842,0] := 73.65, [843,0] := 73.65, [844,0] := 73.65, [845,0] := 73.725, [846,0] := 73.725, [847,0] := 73.725, [848,0] := 73.725, [849,0] := 73.725, [850,0] := 73.65, [851,0] := 73.65, [852,0] := 73.725, [853,0] := 73.725, [854,0] := 73.725, [855,0] := 73.65, [856,0] := 73.65, [857,0] := 73.65, [858,0] := 73.65, [859,0] := 73.65, [860,0] := 73.65, [861,0] := 73.65, [862,0] := 73.65, [863,0] := 73.65, [864,0] := 73.65, [865,0] := 73.65, [866,0] := 73.65, [867,0] := 73.65, [868,0] := 73.65, [869,0] := 73.65, [870,0] := 73.65, [871,0] := 73.65, [872,0] := 73.65, [873,0] := 73.65, [874,0] := 73.65, [875,0] := 73.65, [876,0] := 73.725, [877,0] := 73.725, [878,0] := 73.725, [879,0] := 73.725, [880,0] := 73.725, [881,0] := 73.65, [882,0] := 73.65, [883,0] := 73.65, [884,0] := 73.65, [885,0] := 73.65, [886,0] := 73.65, [887,0] := 73.65, [888,0] := 73.65, [889,0] := 73.65, [890,0] := 73.65, [891,0] := 73.65, [892,0] := 73.65, [893,0] := 73.65, [894,0] := 73.65, [895,0] := 73.65, [896,0] := 73.65, [897,0] := 73.65, [898,0] := 73.65, [899,0] := 73.65,
        [900,0] := 73.65, [901,0] := 73.725, [902,0] := 73.725, [903,0] := 73.65, [904,0] := 73.65, [905,0] := 73.65, [906,0] := 73.65, [907,0] := 73.65, [908,0] := 73.725, [909,0] := 73.725, [910,0] := 73.725, [911,0] := 73.725, [912,0] := 73.725, [913,0] := 73.65, [914,0] := 73.65, [915,0] := 73.65, [916,0] := 73.65, [917,0] := 73.65, [918,0] := 73.65, [919,0] := 73.65, [920,0] := 73.65, [921,0] := 73.65, [922,0] := 73.65, [923,0] := 73.65, [924,0] := 73.65, [925,0] := 73.65, [926,0] := 73.65, [927,0] := 73.65, [928,0] := 73.65, [929,0] := 73.65, [930,0] := 73.65, [931,0] := 73.65, [932,0] := 73.725, [933,0] := 73.725, [934,0] := 73.725, [935,0] := 73.725, [936,0] := 73.725, [937,0] := 73.65, [938,0] := 73.65, [939,0] := 73.65, [940,0] := 73.65, [941,0] := 73.65, [942,0] := 73.65, [943,0] := 73.65, [944,0] := 73.65, [945,0] := 73.65, [946,0] := 73.65, [947,0] := 73.65, [948,0] := 73.65, [949,0] := 73.65, [950,0] := 73.65, [951,0] := 73.65, [952,0] := 73.65, [953,0] := 73.65, [954,0] := 73.65, [955,0] := 73.65, [956,0] := 73.65, [957,0] := 73.65, [958,0] := 73.65, [959,0] := 73.65,
        [960,0] := 73.65, [961,0] := 73.65, [962,0] := 73.65, [963,0] := 73.725, [964,0] := 73.725, [965,0] := 73.725, [966,0] := 73.725, [967,0] := 73.725, [968,0] := 73.65, [969,0] := 73.65, [970,0] := 73.725, [971,0] := 73.725, [972,0] := 73.725, [973,0] := 73.725, [974,0] := 73.725, [975,0] := 73.65, [976,0] := 73.65, [977,0] := 73.65, [978,0] := 73.65, [979,0] := 73.65, [980,0] := 73.65, [981,0] := 73.65, [982,0] := 73.65, [983,0] := 73.65, [984,0] := 73.65, [985,0] := 73.65, [986,0] := 73.65, [987,0] := 73.65, [988,0] := 73.65, [989,0] := 73.65, [990,0] := 73.65, [991,0] := 73.65, [992,0] := 73.65, [993,0] := 73.65, [994,0] := 73.725, [995,0] := 73.725, [996,0] := 73.725, [997,0] := 73.65, [998,0] := 73.65);   // 1000 length 2D FIFO array with flow values and status bits indicating if values have been analysed (1) or not (0) by measCalc()
   FlowArrMem : REAL[1000,2];
   flowCalcOn : BOOL;
   FlowImax : REAL := 18987.0;   // max insp flow in l/min
   FlowImaxArr : REAL[50];   // 50 length array with max insp flow in l/min, from measCalc()
   FlowImaxValue : AOI_Max := (Out_Max := 18987.0, _i := 196);
   FlowO2 : REAL[1000,2] := ([0,0] := 73.8, [1,0] := 73.8, [2,0] := 73.8, [3,0] := 73.8, [4,0] := 73.8, [5,0] := 73.8, [6,0] := 73.8, [7,0] := 73.725, [8,0] := 73.725, [9,0] := 73.725, [10,0] := 73.8, [11,0] := 73.8, [12,0] := 73.8, [13,0] := 73.8, [14,0] := 73.725, [15,0] := 73.725, [16,0] := 73.725, [17,0] := 73.875, [18,0] := 73.875, [19,0] := 73.8, [20,0] := 73.8, [21,0] := 73.8, [22,0] := 73.725, [23,0] := 73.725, [24,0] := 73.8, [25,0] := 73.8, [26,0] := 73.8, [27,0] := 73.8, [28,0] := 73.8, [29,0] := 73.8, [30,0] := 73.8, [31,0] := 73.725, [32,0] := 73.725, [33,0] := 73.725, [34,0] := 73.8, [35,0] := 73.8, [36,0] := 73.8, [37,0] := 73.8, [38,0] := 73.8, [39,0] := 73.725, [40,0] := 73.725, [41,0] := 73.8, [42,0] := 73.8, [43,0] := 73.8, [44,0] := 73.8, [45,0] := 73.8, [46,0] := 73.725, [47,0] := 73.725, [48,0] := 73.8, [49,0] := 73.8, [50,0] := 73.8, [51,0] := 73.8, [52,0] := 73.8, [53,0] := 73.8, [54,0] := 73.8, [55,0] := 73.725, [56,0] := 73.725, [57,0] := 73.725, [58,0] := 73.8, [59,0] := 73.8,
        [60,0] := 73.8, [61,0] := 73.8, [62,0] := 73.8, [63,0] := 73.725, [64,0] := 73.725, [65,0] := 73.875, [66,0] := 73.875, [67,0] := 73.8, [68,0] := 73.8, [69,0] := 73.8, [70,0] := 73.725, [71,0] := 73.725, [72,0] := 73.8, [73,0] := 73.8, [74,0] := 73.8, [75,0] := 73.8, [76,0] := 73.8, [77,0] := 73.725, [78,0] := 73.725, [79,0] := 73.725, [80,0] := 73.8, [81,0] := 73.8, [82,0] := 73.8, [83,0] := 73.8, [84,0] := 73.8, [85,0] := 73.8, [86,0] := 73.8, [87,0] := 73.725, [88,0] := 73.725, [89,0] := 73.8, [90,0] := 73.8, [91,0] := 73.8, [92,0] := 73.8, [93,0] := 73.8, [94,0] := 73.725, [95,0] := 73.725, [96,0] := 73.8, [97,0] := 73.8, [98,0] := 73.8, [99,0] := 73.8, [100,0] := 73.8, [101,0] := 73.725, [102,0] := 73.725, [103,0] := 73.8, [104,0] := 73.8, [105,0] := 73.8, [106,0] := 73.8, [107,0] := 73.8, [108,0] := 73.725, [109,0] := 73.725, [110,0] := 73.725, [111,0] := 73.8, [112,0] := 73.8, [113,0] := 73.8, [114,0] := 73.8, [115,0] := 73.8, [116,0] := 73.8, [117,0] := 73.8, [118,0] := 73.725, [119,0] := 73.725,
        [120,0] := 73.8, [121,0] := 73.8, [122,0] := 73.8, [123,0] := 73.8, [124,0] := 73.8, [125,0] := 73.725, [126,0] := 73.725, [127,0] := 73.725, [128,0] := 73.8, [129,0] := 73.8, [130,0] := 73.8, [131,0] := 73.8, [132,0] := 73.725, [133,0] := 73.725, [134,0] := 73.725, [135,0] := 73.8, [136,0] := 73.8, [137,0] := 73.8, [138,0] := 73.8, [139,0] := 73.8, [140,0] := 73.8, [141,0] := 73.8, [142,0] := 73.725, [143,0] := 73.725, [144,0] := 73.725, [145,0] := 73.8, [146,0] := 73.8, [147,0] := 73.8, [148,0] := 73.8, [149,0] := 73.725, [150,0] := 73.725, [151,0] := 73.725, [152,0] := 73.875, [153,0] := 73.875, [154,0] := 73.8, [155,0] := 73.8, [156,0] := 73.725, [157,0] := 73.725, [158,0] := 73.725, [159,0] := 73.8, [160,0] := 73.8, [161,0] := 73.8, [162,0] := 73.8, [163,0] := 73.8, [164,0] := 73.8, [165,0] := 73.8, [166,0] := 73.725, [167,0] := 73.725, [168,0] := 73.725, [169,0] := 73.8, [170,0] := 73.8, [171,0] := 73.8, [172,0] := 73.8, [173,0] := 73.725, [174,0] := 73.725, [175,0] := 73.725, [176,0] := 73.8, [177,0] := 73.8, [178,0] := 73.8, [179,0] := 73.8,
        [180,0] := 73.8, [181,0] := 73.725, [182,0] := 73.725, [183,0] := 73.8, [184,0] := 73.8, [185,0] := 73.8, [186,0] := 73.8, [187,0] := 73.8, [188,0] := 73.725, [189,0] := 73.725, [190,0] := 73.8, [191,0] := 73.8, [192,0] := 73.8, [193,0] := 73.8, [194,0] := 73.8, [195,0] := 73.8, [196,0] := 73.8, [197,0] := 73.725, [198,0] := 73.725, [199,0] := 73.725, [200,0] := 73.8, [201,0] := 73.8, [202,0] := 73.8, [203,0] := 73.8, [204,0] := 73.8, [205,0] := 73.725, [206,0] := 73.725, [207,0] := 73.875, [208,0] := 73.875, [209,0] := 73.8, [210,0] := 73.8, [211,0] := 73.8, [212,0] := 73.725, [213,0] := 73.725, [214,0] := 73.8, [215,0] := 73.8, [216,0] := 73.8, [217,0] := 73.8, [218,0] := 73.8, [219,0] := 73.8, [220,0] := 73.8, [221,0] := 73.8, [222,0] := 73.8, [223,0] := 73.8, [224,0] := 73.8, [225,0] := 73.8, [226,0] := 73.8, [227,0] := 73.8, [228,0] := 73.8, [229,0] := 73.725, [230,0] := 73.725, [231,0] := 73.8, [232,0] := 73.8, [233,0] := 73.8, [234,0] := 73.8, [235,0] := 73.8, [236,0] := 73.725, [237,0] := 73.725, [238,0] := 73.875, [239,0] := 73.875,
        [240,0] := 73.875, [241,0] := 73.8, [242,0] := 73.8, [243,0] := 73.725, [244,0] := 73.725, [245,0] := 73.725, [246,0] := 73.8, [247,0] := 73.8, [248,0] := 73.8, [249,0] := 73.8, [250,0] := 73.8, [251,0] := 73.8, [252,0] := 73.8, [253,0] := 73.8, [254,0] := 73.8, [255,0] := 73.8, [256,0] := 73.8, [257,0] := 73.8, [258,0] := 73.8, [259,0] := 73.8, [260,0] := 73.725, [261,0] := 73.725, [262,0] := 73.875, [263,0] := 73.875, [264,0] := 73.875, [265,0] := 73.8, [266,0] := 73.8, [267,0] := 73.725, [268,0] := 73.725, [269,0] := 73.725, [270,0] := 73.8, [271,0] := 73.8, [272,0] := 73.8, [273,0] := 73.8, [274,0] := 73.725, [275,0] := 73.725, [276,0] := 73.725, [277,0] := 73.725, [278,0] := 73.725, [279,0] := 73.8, [280,0] := 73.8, [281,0] := 73.8, [282,0] := 73.8, [283,0] := 73.8, [284,0] := 73.725, [285,0] := 73.725, [286,0] := 73.725, [287,0] := 73.875, [288,0] := 73.875, [289,0] := 73.8, [290,0] := 73.8, [291,0] := 73.725, [292,0] := 73.725, [293,0] := 73.725, [294,0] := 73.8, [295,0] := 73.8, [296,0] := 73.8, [297,0] := 73.8, [298,0] := 73.8, [299,0] := 73.8,
        [300,0] := 73.8, [301,0] := 73.725, [302,0] := 73.725, [303,0] := 73.8, [304,0] := 73.8, [305,0] := 73.8, [306,0] := 73.8, [307,0] := 73.8, [308,0] := 73.725, [309,0] := 73.725, [310,0] := 73.725, [311,0] := 73.8, [312,0] := 73.8, [313,0] := 73.875, [314,0] := 73.875, [315,0] := 73.875, [316,0] := 73.725, [317,0] := 73.725, [318,0] := 73.8, [319,0] := 73.8, [320,0] := 73.8, [321,0] := 73.8, [322,0] := 73.8, [323,0] := 73.725, [324,0] := 73.725, [325,0] := 73.8, [326,0] := 73.8, [327,0] := 73.8, [328,0] := 73.8, [329,0] := 73.8, [330,0] := 73.8, [331,0] := 73.8, [332,0] := 73.725, [333,0] := 73.725, [334,0] := 73.725, [335,0] := 73.8, [336,0] := 73.8, [337,0] := 73.8, [338,0] := 73.8, [339,0] := 73.8, [340,0] := 73.725, [341,0] := 73.725, [342,0] := 73.875, [343,0] := 73.875, [344,0] := 73.8, [345,0] := 73.8, [346,0] := 73.8, [347,0] := 73.725, [348,0] := 73.725, [349,0] := 73.8, [350,0] := 73.8, [351,0] := 73.8, [352,0] := 73.8, [353,0] := 73.8, [354,0] := 73.8, [355,0] := 73.8, [356,0] := 73.725, [357,0] := 73.725, [358,0] := 73.725, [359,0] := 73.8,
        [360,0] := 73.8, [361,0] := 73.8, [362,0] := 73.8, [363,0] := 73.8, [364,0] := 73.725, [365,0] := 73.725, [366,0] := 73.875, [367,0] := 73.875, [368,0] := 73.8, [369,0] := 73.8, [370,0] := 73.8, [371,0] := 73.725, [372,0] := 73.725, [373,0] := 73.8, [374,0] := 73.8, [375,0] := 73.8, [376,0] := 73.8, [377,0] := 73.8, [378,0] := 73.8, [379,0] := 73.8, [380,0] := 73.8, [381,0] := 73.8, [382,0] := 73.8, [383,0] := 73.8, [384,0] := 73.8, [385,0] := 73.8, [386,0] := 73.8, [387,0] := 73.8, [388,0] := 73.725, [389,0] := 73.725, [390,0] := 73.8, [391,0] := 73.8, [392,0] := 73.8, [393,0] := 73.8, [394,0] := 73.8, [395,0] := 73.725, [396,0] := 73.725, [397,0] := 73.8, [398,0] := 73.8, [399,0] := 73.8, [400,0] := 73.8, [401,0] := 73.8, [402,0] := 73.725, [403,0] := 73.725, [404,0] := 73.725, [405,0] := 73.8, [406,0] := 73.8, [407,0] := 73.8, [408,0] := 73.8, [409,0] := 73.8, [410,0] := 73.8, [411,0] := 73.8, [412,0] := 73.725, [413,0] := 73.725, [414,0] := 73.8, [415,0] := 73.8, [416,0] := 73.8, [417,0] := 73.8, [418,0] := 73.8, [419,0] := 73.725,
        [420,0] := 73.725, [421,0] := 73.875, [422,0] := 73.875, [423,0] := 73.875, [424,0] := 73.8, [425,0] := 73.8, [426,0] := 73.725, [427,0] := 73.725, [428,0] := 73.725, [429,0] := 73.8, [430,0] := 73.8, [431,0] := 73.8, [432,0] := 73.8, [433,0] := 73.8, [434,0] := 73.8, [435,0] := 73.8, [436,0] := 73.8, [437,0] := 73.8, [438,0] := 73.8, [439,0] := 73.8, [440,0] := 73.8, [441,0] := 73.8, [442,0] := 73.8, [443,0] := 73.725, [444,0] := 73.725, [445,0] := 73.725, [446,0] := 73.8, [447,0] := 73.8, [448,0] := 73.8, [449,0] := 73.8, [450,0] := 73.725, [451,0] := 73.725, [452,0] := 73.725, [453,0] := 73.875, [454,0] := 73.875, [455,0] := 73.875, [456,0] := 73.875, [457,0] := 73.725, [458,0] := 73.725, [459,0] := 73.725, [460,0] := 73.8, [461,0] := 73.8, [462,0] := 73.8, [463,0] := 73.8, [464,0] := 73.8, [465,0] := 73.725, [466,0] := 73.725, [467,0] := 73.725, [468,0] := 73.725, [469,0] := 73.725, [470,0] := 73.8, [471,0] := 73.8, [472,0] := 73.8, [473,0] := 73.8, [474,0] := 73.725, [475,0] := 73.725, [476,0] := 73.725, [477,0] := 73.8, [478,0] := 73.8, [479,0] := 73.8,
        [480,0] := 73.8, [481,0] := 73.8, [482,0] := 73.725, [483,0] := 73.725, [484,0] := 73.8, [485,0] := 73.8, [486,0] := 73.8, [487,0] := 73.8, [488,0] := 73.8, [489,0] := 73.725, [490,0] := 73.725, [491,0] := 73.8, [492,0] := 73.8, [493,0] := 73.8, [494,0] := 73.8, [495,0] := 73.8, [496,0] := 73.8, [497,0] := 73.8, [498,0] := 73.725, [499,0] := 73.725, [500,0] := 73.725, [501,0] := 73.8, [502,0] := 73.8, [503,0] := 73.8, [504,0] := 73.8, [505,0] := 73.8, [506,0] := 73.725, [507,0] := 73.725, [508,0] := 73.875, [509,0] := 73.875, [510,0] := 73.875, [511,0] := 73.8, [512,0] := 73.8, [513,0] := 73.725, [514,0] := 73.725, [515,0] := 73.8, [516,0] := 73.8, [517,0] := 73.8, [518,0] := 73.8, [519,0] := 73.8, [520,0] := 73.725, [521,0] := 73.725, [522,0] := 73.8, [523,0] := 73.8, [524,0] := 73.8, [525,0] := 73.8, [526,0] := 73.8, [527,0] := 73.8, [528,0] := 73.8, [529,0] := 73.8, [530,0] := 73.725, [531,0] := 73.725, [532,0] := 73.8, [533,0] := 73.8, [534,0] := 73.8, [535,0] := 73.8, [536,0] := 73.8, [537,0] := 73.725, [538,0] := 73.725, [539,0] := 73.875,
        [540,0] := 73.875, [541,0] := 73.875, [542,0] := 73.8, [543,0] := 73.8, [544,0] := 73.725, [545,0] := 73.725, [546,0] := 73.725, [547,0] := 73.8, [548,0] := 73.8, [549,0] := 73.8, [550,0] := 73.8, [551,0] := 73.725, [552,0] := 73.725, [553,0] := 73.725, [554,0] := 73.8, [555,0] := 73.8, [556,0] := 73.8, [557,0] := 73.8, [558,0] := 73.8, [559,0] := 73.8, [560,0] := 73.8, [561,0] := 73.725, [562,0] := 73.725, [563,0] := 73.8, [564,0] := 73.8, [565,0] := 73.8, [566,0] := 73.8, [567,0] := 73.8, [568,0] := 73.725, [569,0] := 73.725, [570,0] := 73.875, [571,0] := 73.875, [572,0] := 73.875, [573,0] := 73.8, [574,0] := 73.8, [575,0] := 73.725, [576,0] := 73.725, [577,0] := 73.725, [578,0] := 73.8, [579,0] := 73.8, [580,0] := 73.8, [581,0] := 73.8, [582,0] := 73.8, [583,0] := 73.725, [584,0] := 73.725, [585,0] := 73.8, [586,0] := 73.8, [587,0] := 73.8, [588,0] := 73.8, [589,0] := 73.8, [590,0] := 73.8, [591,0] := 73.8, [592,0] := 73.725, [593,0] := 73.725, [594,0] := 73.725, [595,0] := 73.8, [596,0] := 73.8, [597,0] := 73.8, [598,0] := 73.8, [599,0] := 73.8,
        [600,0] := 73.725, [601,0] := 73.725, [602,0] := 73.8, [603,0] := 73.8, [604,0] := 73.8, [605,0] := 73.8, [606,0] := 73.8, [607,0] := 73.8, [608,0] := 73.8, [609,0] := 73.8, [610,0] := 73.8, [611,0] := 73.8, [612,0] := 73.8, [613,0] := 73.8, [614,0] := 73.8, [615,0] := 73.8, [616,0] := 73.725, [617,0] := 73.725, [618,0] := 73.725, [619,0] := 73.8, [620,0] := 73.8, [621,0] := 73.8, [622,0] := 73.8, [623,0] := 73.8, [624,0] := 73.725, [625,0] := 73.725, [626,0] := 73.875, [627,0] := 73.875, [628,0] := 73.8, [629,0] := 73.8, [630,0] := 73.8, [631,0] := 73.725, [632,0] := 73.725, [633,0] := 73.725, [634,0] := 73.725, [635,0] := 73.725, [636,0] := 73.8, [637,0] := 73.8, [638,0] := 73.8, [639,0] := 73.8, [640,0] := 73.725, [641,0] := 73.725, [642,0] := 73.725, [643,0] := 73.875, [644,0] := 73.875, [645,0] := 73.8, [646,0] := 73.8, [647,0] := 73.8, [648,0] := 73.725, [649,0] := 73.725, [650,0] := 73.8, [651,0] := 73.8, [652,0] := 73.8, [653,0] := 73.8, [654,0] := 73.8, [655,0] := 73.725, [656,0] := 73.725, [657,0] := 73.8, [658,0] := 73.8, [659,0] := 73.8,
        [660,0] := 73.8, [661,0] := 73.8, [662,0] := 73.8, [663,0] := 73.8, [664,0] := 73.725, [665,0] := 73.725, [666,0] := 73.725, [667,0] := 73.8, [668,0] := 73.8, [669,0] := 73.8, [670,0] := 73.8, [671,0] := 73.8, [672,0] := 73.725, [673,0] := 73.725, [674,0] := 73.875, [675,0] := 73.875, [676,0] := 73.875, [677,0] := 73.8, [678,0] := 73.8, [679,0] := 73.725, [680,0] := 73.725, [681,0] := 73.8, [682,0] := 73.8, [683,0] := 73.8, [684,0] := 73.8, [685,0] := 73.8, [686,0] := 73.8, [687,0] := 73.8, [688,0] := 73.8, [689,0] := 73.725, [690,0] := 73.725, [691,0] := 73.8, [692,0] := 73.8, [693,0] := 73.8, [694,0] := 73.8, [695,0] := 73.8, [696,0] := 73.725, [697,0] := 73.725, [698,0] := 73.8, [699,0] := 73.8, [700,0] := 73.8, [701,0] := 73.8, [702,0] := 73.8, [703,0] := 73.725, [704,0] := 73.725, [705,0] := 73.8, [706,0] := 73.8, [707,0] := 73.8, [708,0] := 73.8, [709,0] := 73.8, [710,0] := 73.725, [711,0] := 73.725, [712,0] := 73.725, [713,0] := 73.8, [714,0] := 73.8, [715,0] := 73.8, [716,0] := 73.8, [717,0] := 73.8, [718,0] := 73.8, [719,0] := 73.8,
        [720,0] := 73.725, [721,0] := 73.725, [722,0] := 73.8, [723,0] := 73.8, [724,0] := 73.8, [725,0] := 73.8, [726,0] := 73.8, [727,0] := 73.725, [728,0] := 73.725, [729,0] := 73.725, [730,0] := 73.875, [731,0] := 73.875, [732,0] := 73.8, [733,0] := 73.8, [734,0] := 73.725, [735,0] := 73.725, [736,0] := 73.725, [737,0] := 73.8, [738,0] := 73.8, [739,0] := 73.8, [740,0] := 73.8, [741,0] := 73.8, [742,0] := 73.8, [743,0] := 73.8, [744,0] := 73.725, [745,0] := 73.725, [746,0] := 73.8, [747,0] := 73.8, [748,0] := 73.8, [749,0] := 73.8, [750,0] := 73.8, [751,0] := 73.725, [752,0] := 73.725, [753,0] := 73.725, [754,0] := 73.875, [755,0] := 73.875, [756,0] := 73.8, [757,0] := 73.8, [758,0] := 73.725, [759,0] := 73.725, [760,0] := 73.725, [761,0] := 73.8, [762,0] := 73.8, [763,0] := 73.8, [764,0] := 73.8, [765,0] := 73.8, [766,0] := 73.725, [767,0] := 73.725, [768,0] := 73.8, [769,0] := 73.8, [770,0] := 73.8, [771,0] := 73.8, [772,0] := 73.8, [773,0] := 73.8, [774,0] := 73.8, [775,0] := 73.725, [776,0] := 73.725, [777,0] := 73.725, [778,0] := 73.8, [779,0] := 73.8,
        [780,0] := 73.8, [781,0] := 73.8, [782,0] := 73.725, [783,0] := 73.725, [784,0] := 73.725, [785,0] := 73.8, [786,0] := 73.8, [787,0] := 73.8, [788,0] := 73.8, [789,0] := 73.8, [790,0] := 73.725, [791,0] := 73.725, [792,0] := 73.8, [793,0] := 73.8, [794,0] := 73.8, [795,0] := 73.8, [796,0] := 73.8, [797,0] := 73.8, [798,0] := 73.8, [799,0] := 73.725, [800,0] := 73.725, [801,0] := 73.725, [802,0] := 73.8, [803,0] := 73.8, [804,0] := 73.8, [805,0] := 73.8, [806,0] := 73.8, [807,0] := 73.725, [808,0] := 73.725, [809,0] := 73.875, [810,0] := 73.875, [811,0] := 73.875, [812,0] := 73.875, [813,0] := 73.875, [814,0] := 73.725, [815,0] := 73.725, [816,0] := 73.8, [817,0] := 73.8, [818,0] := 73.8, [819,0] := 73.8, [820,0] := 73.8, [821,0] := 73.8, [822,0] := 73.8, [823,0] := 73.725, [824,0] := 73.725, [825,0] := 73.725, [826,0] := 73.8, [827,0] := 73.8, [828,0] := 73.8, [829,0] := 73.8, [830,0] := 73.8, [831,0] := 73.725, [832,0] := 73.725, [833,0] := 73.8, [834,0] := 73.8, [835,0] := 73.8, [836,0] := 73.8, [837,0] := 73.8, [838,0] := 73.725, [839,0] := 73.725,
        [840,0] := 73.8, [841,0] := 73.8, [842,0] := 73.8, [843,0] := 73.8, [844,0] := 73.8, [845,0] := 73.725, [846,0] := 73.725, [847,0] := 73.725, [848,0] := 73.8, [849,0] := 73.8, [850,0] := 73.8, [851,0] := 73.8, [852,0] := 73.8, [853,0] := 73.8, [854,0] := 73.8, [855,0] := 73.725, [856,0] := 73.725, [857,0] := 73.8, [858,0] := 73.8, [859,0] := 73.8, [860,0] := 73.8, [861,0] := 73.8, [862,0] := 73.725, [863,0] := 73.725, [864,0] := 73.725, [865,0] := 73.8, [866,0] := 73.8, [867,0] := 73.8, [868,0] := 73.8, [869,0] := 73.725, [870,0] := 73.725, [871,0] := 73.725, [872,0] := 73.725, [873,0] := 73.725, [874,0] := 73.8, [875,0] := 73.8, [876,0] := 73.8, [877,0] := 73.8, [878,0] := 73.725, [879,0] := 73.725, [880,0] := 73.725, [881,0] := 73.875, [882,0] := 73.875, [883,0] := 73.8, [884,0] := 73.8, [885,0] := 73.8, [886,0] := 73.725, [887,0] := 73.725, [888,0] := 73.8, [889,0] := 73.8, [890,0] := 73.8, [891,0] := 73.8, [892,0] := 73.8, [893,0] := 73.725, [894,0] := 73.725, [895,0] := 73.8, [896,0] := 73.8, [897,0] := 73.8, [898,0] := 73.8, [899,0] := 73.8,
        [900,0] := 73.8, [901,0] := 73.8, [902,0] := 73.8, [903,0] := 73.725, [904,0] := 73.725, [905,0] := 73.8, [906,0] := 73.8, [907,0] := 73.8, [908,0] := 73.8, [909,0] := 73.8, [910,0] := 73.725, [911,0] := 73.725, [912,0] := 73.875, [913,0] := 73.875, [914,0] := 73.875, [915,0] := 73.8, [916,0] := 73.8, [917,0] := 73.725, [918,0] := 73.725, [919,0] := 73.725, [920,0] := 73.8, [921,0] := 73.8, [922,0] := 73.8, [923,0] := 73.8, [924,0] := 73.725, [925,0] := 73.725, [926,0] := 73.725, [927,0] := 73.8, [928,0] := 73.8, [929,0] := 73.8, [930,0] := 73.8, [931,0] := 73.8, [932,0] := 73.8, [933,0] := 73.8, [934,0] := 73.725, [935,0] := 73.725, [936,0] := 73.875, [937,0] := 73.875, [938,0] := 73.875, [939,0] := 73.8, [940,0] := 73.8, [941,0] := 73.725, [942,0] := 73.725, [943,0] := 73.725, [944,0] := 73.8, [945,0] := 73.8, [946,0] := 73.8, [947,0] := 73.8, [948,0] := 73.725, [949,0] := 73.725, [950,0] := 73.725, [951,0] := 73.8, [952,0] := 73.8, [953,0] := 73.8, [954,0] := 73.8, [955,0] := 73.8, [956,0] := 73.8, [957,0] := 73.8, [958,0] := 73.725, [959,0] := 73.725,
        [960,0] := 73.8, [961,0] := 73.8, [962,0] := 73.8, [963,0] := 73.8, [964,0] := 73.8, [965,0] := 73.725, [966,0] := 73.725, [967,0] := 73.725, [968,0] := 73.8, [969,0] := 73.8, [970,0] := 73.8, [971,0] := 73.8, [972,0] := 73.8, [973,0] := 73.8, [974,0] := 73.8, [975,0] := 73.725, [976,0] := 73.725, [977,0] := 73.8, [978,0] := 73.8, [979,0] := 73.8, [980,0] := 73.8, [981,0] := 73.8, [982,0] := 73.725, [983,0] := 73.725, [984,0] := 73.875, [985,0] := 73.875, [986,0] := 73.875, [987,0] := 73.875, [988,0] := 73.875, [989,0] := 73.725, [990,0] := 73.725, [991,0] := 73.725, [992,0] := 73.875, [993,0] := 73.875, [994,0] := 73.8, [995,0] := 73.8, [996,0] := 73.8, [997,0] := 73.725, [998,0] := 73.725);
   FlowO2Mem : REAL[1000,2];
   FractionAir : REAL := 0.94936705;
   FractionO2 : REAL := 0.050632954;
   GetSlaveValue : MOTION_INSTRUCTION := (FLAGS := -1577058304, EN := 1, DN := 1);
   HMI_ScreenNo : DINT;
   HMIStart : BOOL;
   HMIStop : BOOL;
   i : DINT := 101;
   I_E : STRING := '1:3';   // part of I:E ratio: 1, 2, 3 or 4
   IE : STRING[4] := ([0] := '1:1', [1] := '1:2', [2] := '1:3', [3] := '1:4');
   IE_counter : DINT := 2;
   IE_E : INT := 3;
   IE_ERunning : INT := 3;
   IE_I : INT := 1;
   IE_IRunning : INT := 1;
   Insp : BOOL := 1;
   inspAirFlowCtrl : REAL[650] := ([1] := 3.4177215, [2] := 6.835443, [3] := 10.253164, [4] := 13.670886, [5] := 17.088608, [6] := 20.506329, [7] := 23.924051, [8] := 27.341772, [9] := 30.759493, [10] := 34.177216, [11] := 37.594936, [12] := 41.012657, [13] := 44.430378, [14] := 47.848103, [15] := 51.265823, [16] := 54.683544, [17] := 58.101265, [18] := 61.518986, [19] := 64.93671, [20] := 68.35443, [21] := 68.35443, [22] := 68.35443, [23] := 68.35443, [24] := 68.35443, [25] := 68.35443, [26] := 68.35443, [27] := 68.35443, [28] := 68.35443, [29] := 68.35443, [30] := 68.35443, [31] := 68.35443, [32] := 68.35443, [33] := 68.35443, [34] := 68.35443, [35] := 68.35443, [36] := 68.35443, [37] := 68.35443, [38] := 68.35443, [39] := 68.35443, [40] := 68.35443, [41] := 68.35443, [42] := 68.35443, [43] := 68.35443, [44] := 68.35443, [45] := 68.35443, [46] := 68.35443, [47] := 68.35443, [48] := 68.35443, [49] := 68.35443, [50] := 68.35443, [51] := 68.35443, [52] := 68.35443, [53] := 68.35443, [54] := 68.35443, [55] := 68.35443, [56] := 68.35443, [57] := 68.35443, [58] := 68.35443, [59] := 68.35443);   // 650 length array with flow values for insp air valve, moved from nextInspAirFlowCtrl[] by ISR_ValveCtrl()
   inspAirFlowCtrlNew : REAL[650] := ([1] := 3.4177215, [2] := 6.835443, [3] := 10.253164, [4] := 13.670886, [5] := 17.088608, [6] := 20.506329, [7] := 23.924051, [8] := 27.341772, [9] := 30.759493, [10] := 34.177216, [11] := 37.594936, [12] := 41.012657, [13] := 44.430378, [14] := 47.848103, [15] := 51.265823, [16] := 54.683544, [17] := 58.101265, [18] := 61.518986, [19] := 64.93671, [20] := 68.35443, [21] := 68.35443, [22] := 68.35443, [23] := 68.35443, [24] := 68.35443, [25] := 68.35443, [26] := 68.35443, [27] := 68.35443, [28] := 68.35443, [29] := 68.35443, [30] := 68.35443, [31] := 68.35443, [32] := 68.35443, [33] := 68.35443, [34] := 68.35443, [35] := 68.35443, [36] := 68.35443, [37] := 68.35443, [38] := 68.35443, [39] := 68.35443, [40] := 68.35443, [41] := 68.35443, [42] := 68.35443, [43] := 68.35443, [44] := 68.35443, [45] := 68.35443, [46] := 68.35443, [47] := 68.35443, [48] := 68.35443, [49] := 68.35443, [50] := 68.35443, [51] := 68.35443, [52] := 68.35443, [53] := 68.35443, [54] := 68.35443, [55] := 68.35443, [56] := 68.35443, [57] := 68.35443, [58] := 68.35443, [59] := 68.35443);
   inspCount : INT;   // between 1-650 to indicate where valveCtrl should read from inspAirFlowCtrl[] and inspO2FlowCtrl[]
   inspCountLength : INT := 100;   // between 1-650 to indicate when valveCtrl should stop reading from inspAirFlowCtrl[] and inspO2FlowCtrl[], copied from nextInspCountLength by ISR_ValveCtrl()
   inspCountLengthNew : REAL := 100.0;
   inspCounts : REAL := 100.00001;
   inspExp : BOOL;   // 1: inspiration, 0: expiration
   InspiratoryRampTimeInMS : REAL := 200.00002;
   inspO2FlowCtrl : REAL[650] := ([1] := 0.18227863, [2] := 0.36455727, [3] := 0.5468359, [4] := 0.72911453, [5] := 0.91139317, [6] := 1.0936718, [7] := 1.2759504, [8] := 1.4582291, [9] := 1.6405077, [10] := 1.8227863, [11] := 2.005065, [12] := 2.1873436, [13] := 2.3696222, [14] := 2.5519009, [15] := 2.7341795, [16] := 2.9164581, [17] := 3.0987368, [18] := 3.2810154, [19] := 3.463294, [20] := 3.6455727, [21] := 3.6455727, [22] := 3.6455727, [23] := 3.6455727, [24] := 3.6455727, [25] := 3.6455727, [26] := 3.6455727, [27] := 3.6455727, [28] := 3.6455727, [29] := 3.6455727, [30] := 3.6455727, [31] := 3.6455727, [32] := 3.6455727, [33] := 3.6455727, [34] := 3.6455727, [35] := 3.6455727, [36] := 3.6455727, [37] := 3.6455727, [38] := 3.6455727, [39] := 3.6455727, [40] := 3.6455727, [41] := 3.6455727, [42] := 3.6455727, [43] := 3.6455727, [44] := 3.6455727, [45] := 3.6455727, [46] := 3.6455727, [47] := 3.6455727, [48] := 3.6455727, [49] := 3.6455727, [50] := 3.6455727, [51] := 3.6455727, [52] := 3.6455727, [53] := 3.6455727, [54] := 3.6455727, [55] := 3.6455727, [56] := 3.6455727, [57] := 3.6455727, [58] := 3.6455727, [59] := 3.6455727);   // 650 length array with flow values for insp O2 valve, moved from nextInspO2FlowCtrl[] by ISR_ValveCtrl()
   inspO2FlowCtrlNew : REAL[650] := ([1] := 0.18227863, [2] := 0.36455727, [3] := 0.5468359, [4] := 0.72911453, [5] := 0.91139317, [6] := 1.0936718, [7] := 1.2759504, [8] := 1.4582291, [9] := 1.6405077, [10] := 1.8227863, [11] := 2.005065, [12] := 2.1873436, [13] := 2.3696222, [14] := 2.5519009, [15] := 2.7341795, [16] := 2.9164581, [17] := 3.0987368, [18] := 3.2810154, [19] := 3.463294, [20] := 3.6455727, [21] := 3.6455727, [22] := 3.6455727, [23] := 3.6455727, [24] := 3.6455727, [25] := 3.6455727, [26] := 3.6455727, [27] := 3.6455727, [28] := 3.6455727, [29] := 3.6455727, [30] := 3.6455727, [31] := 3.6455727, [32] := 3.6455727, [33] := 3.6455727, [34] := 3.6455727, [35] := 3.6455727, [36] := 3.6455727, [37] := 3.6455727, [38] := 3.6455727, [39] := 3.6455727, [40] := 3.6455727, [41] := 3.6455727, [42] := 3.6455727, [43] := 3.6455727, [44] := 3.6455727, [45] := 3.6455727, [46] := 3.6455727, [47] := 3.6455727, [48] := 3.6455727, [49] := 3.6455727, [50] := 3.6455727, [51] := 3.6455727, [52] := 3.6455727, [53] := 3.6455727, [54] := 3.6455727, [55] := 3.6455727, [56] := 3.6455727, [57] := 3.6455727, [58] := 3.6455727, [59] := 3.6455727);
   inspPauseCalc : REAL := 40.000004;
   inspPauseNrOfAdjustments : REAL := 40.0;
   inspPauseStartI : INT;
   inspPauseTime : INT := 10;
   inspPauseTimeInMS : REAL := 400.00003;
   inspPauseTimePercent : REAL := 0.1;
   inspPauseTimeRunning : INT := 10;
   inspRampTime : INT := 5;
   inspRampTimePercent : REAL := 0.05;
   inspRampTimeRunning : INT := 5;
   inspStartI : INT;
   inspTimeinMS : REAL := 1000.00006;
   last_state : DINT := 3;
   maxFlowAllowed : INT := 100;
   Mean50 : AOI_Mean50 := (In_N0 := 1, Out_Mean := 2.059567, _i := 2);
   MeanFilter : AOI_FilterSignal;
   message : STRING := 'Data Ready';
   Messages_to_user : STRING[10] := ([0] := 'Data Ready', [1] := 'Length of Insp or Exp is wrong', [2] := 'Insp Flow too high for sensor');
   Mode : STRING := 'VC';
   ModeOptions : STRING[4];
   MV : REAL := 48025.97;   // minute ventilation in l/min
   MVArr : REAL[50];   // 50 length array with minute ventilation in l/min, from measCalc()
   NewBreath : BOOL;   // 1:set by BreathDetect() to signal that full not previously analysed insp data set available
   NewExpOpenCloseAvail : BOOL;   // signal to valveCtrl to include new expOpenCloseCtrl[]to overwrite when expiration ended, set by calcBreath()
   newInspFlowAvil : BOOL;
   NewSettings : BOOL;
   NewTimeRate_p5 : DINT := 10000;
   NewTimeRate_p8 : DINT := 10000;
   nextExpCountLength : INT := 300;   // between 1-1000 to indicate when valveCtrl should stop reading from expOpenCloseCtrl[], set by calcBreath()
   nextExpOpenCloseCtrl : INT[1000] := ([0] := 1, [1] := 1, [2] := 1, [3] := 1, [4] := 1, [5] := 1, [6] := 1, [7] := 1, [8] := 1, [9] := 1, [10] := 1, [11] := 1, [12] := 1, [13] := 1, [14] := 1, [15] := 1, [16] := 1, [17] := 1, [18] := 1, [19] := 1, [20] := 1, [21] := 1, [22] := 1, [23] := 1, [24] := 1, [25] := 1, [26] := 1, [27] := 1, [28] := 1, [29] := 1, [30] := 1, [31] := 1, [32] := 1, [33] := 1, [34] := 1, [35] := 1, [36] := 1, [37] := 1, [38] := 1, [39] := 1, [40] := 1, [41] := 1, [42] := 1, [43] := 1, [44] := 1, [45] := 1, [46] := 1, [47] := 1, [48] := 1, [49] := 1, [50] := 1, [51] := 1, [52] := 1, [53] := 1, [54] := 1, [55] := 1, [56] := 1, [57] := 1, [58] := 1, [59] := 1,
        [60] := 1, [61] := 1, [62] := 1, [63] := 1, [64] := 1, [65] := 1, [66] := 1, [67] := 1, [68] := 1, [69] := 1, [70] := 1, [71] := 1, [72] := 1, [73] := 1, [74] := 1, [75] := 1, [76] := 1, [77] := 1, [78] := 1, [79] := 1, [80] := 1, [81] := 1, [82] := 1, [83] := 1, [84] := 1, [85] := 1, [86] := 1, [87] := 1, [88] := 1, [89] := 1, [90] := 1, [91] := 1, [92] := 1, [93] := 1, [94] := 1, [95] := 1, [96] := 1, [97] := 1, [98] := 1, [99] := 1, [100] := 1, [101] := 1, [102] := 1, [103] := 1, [104] := 1, [105] := 1, [106] := 1, [107] := 1, [108] := 1, [109] := 1, [110] := 1, [111] := 1, [112] := 1, [113] := 1, [114] := 1, [115] := 1, [116] := 1, [117] := 1, [118] := 1, [119] := 1,
        [120] := 1, [121] := 1, [122] := 1, [123] := 1, [124] := 1, [125] := 1, [126] := 1, [127] := 1, [128] := 1, [129] := 1, [130] := 1, [131] := 1, [132] := 1, [133] := 1, [134] := 1, [135] := 1, [136] := 1, [137] := 1, [138] := 1, [139] := 1, [140] := 1, [141] := 1, [142] := 1, [143] := 1, [144] := 1, [145] := 1, [146] := 1, [147] := 1, [148] := 1, [149] := 1, [150] := 1, [151] := 1, [152] := 1, [153] := 1, [154] := 1, [155] := 1, [156] := 1, [157] := 1, [158] := 1, [159] := 1, [160] := 1, [161] := 1, [162] := 1, [163] := 1, [164] := 1, [165] := 1, [166] := 1, [167] := 1, [168] := 1, [169] := 1, [170] := 1, [171] := 1, [172] := 1, [173] := 1, [174] := 1, [175] := 1, [176] := 1, [177] := 1, [178] := 1, [179] := 1,
        [180] := 1, [181] := 1, [182] := 1, [183] := 1, [184] := 1, [185] := 1, [186] := 1, [187] := 1, [188] := 1, [189] := 1, [190] := 1, [191] := 1, [192] := 1, [193] := 1, [194] := 1, [195] := 1, [196] := 1, [197] := 1, [198] := 1, [199] := 1, [200] := 1, [201] := 1, [202] := 1, [203] := 1, [204] := 1, [205] := 1, [206] := 1, [207] := 1, [208] := 1, [209] := 1, [210] := 1, [211] := 1, [212] := 1, [213] := 1, [214] := 1, [215] := 1, [216] := 1, [217] := 1, [218] := 1, [219] := 1, [220] := 1, [221] := 1, [222] := 1, [223] := 1, [224] := 1, [225] := 1, [226] := 1, [227] := 1, [228] := 1, [229] := 1, [230] := 1, [231] := 1, [232] := 1, [233] := 1, [234] := 1, [235] := 1, [236] := 1, [237] := 1, [238] := 1, [239] := 1,
        [240] := 1, [241] := 1, [242] := 1, [243] := 1, [244] := 1, [245] := 1, [246] := 1, [247] := 1, [248] := 1, [249] := 1, [250] := 1, [251] := 1, [252] := 1, [253] := 1, [254] := 1, [255] := 1, [256] := 1, [257] := 1, [258] := 1, [259] := 1, [260] := 1, [261] := 1, [262] := 1, [263] := 1, [264] := 1, [265] := 1, [266] := 1, [267] := 1, [268] := 1, [269] := 1, [270] := 1, [271] := 1, [272] := 1, [273] := 1, [274] := 1, [275] := 1, [276] := 1, [277] := 1, [278] := 1, [279] := 1, [280] := 1, [281] := 1, [282] := 1, [283] := 1, [284] := 1, [285] := 1, [286] := 1, [287] := 1, [288] := 1, [289] := 1, [290] := 1, [291] := 1, [292] := 1, [293] := 1, [294] := 1, [295] := 1, [296] := 1, [297] := 1, [298] := 1, [299] := 1);   // 1000 length array with open (1) or close (0) for exp valve, set by calcBreath()
   nextInspAirFlowCtrl : REAL[650] := ([1] := 3.4177215, [2] := 6.835443, [3] := 10.253164, [4] := 13.670886, [5] := 17.088608, [6] := 20.506329, [7] := 23.924051, [8] := 27.341772, [9] := 30.759493, [10] := 34.177216, [11] := 37.594936, [12] := 41.012657, [13] := 44.430378, [14] := 47.848103, [15] := 51.265823, [16] := 54.683544, [17] := 58.101265, [18] := 61.518986, [19] := 64.93671, [20] := 68.35443, [21] := 68.35443, [22] := 68.35443, [23] := 68.35443, [24] := 68.35443, [25] := 68.35443, [26] := 68.35443, [27] := 68.35443, [28] := 68.35443, [29] := 68.35443, [30] := 68.35443, [31] := 68.35443, [32] := 68.35443, [33] := 68.35443, [34] := 68.35443, [35] := 68.35443, [36] := 68.35443, [37] := 68.35443, [38] := 68.35443, [39] := 68.35443, [40] := 68.35443, [41] := 68.35443, [42] := 68.35443, [43] := 68.35443, [44] := 68.35443, [45] := 68.35443, [46] := 68.35443, [47] := 68.35443, [48] := 68.35443, [49] := 68.35443, [50] := 68.35443, [51] := 68.35443, [52] := 68.35443, [53] := 68.35443, [54] := 68.35443, [55] := 68.35443, [56] := 68.35443, [57] := 68.35443, [58] := 68.35443, [59] := 68.35443);   // 650 length array with flow values for insp air valve, set by calcBreath()
   nextInspCountLength : INT := 100;   // between 1-650 to indicate when valveCtrl should stop reading from inspAirFlowCtrl[] and inspO2FlowCtrl[], set by calcBreath()
   nextInspO2FlowCtrl : REAL[650] := ([1] := 0.18227863, [2] := 0.36455727, [3] := 0.5468359, [4] := 0.72911453, [5] := 0.91139317, [6] := 1.0936718, [7] := 1.2759504, [8] := 1.4582291, [9] := 1.6405077, [10] := 1.8227863, [11] := 2.005065, [12] := 2.1873436, [13] := 2.3696222, [14] := 2.5519009, [15] := 2.7341795, [16] := 2.9164581, [17] := 3.0987368, [18] := 3.2810154, [19] := 3.463294, [20] := 3.6455727, [21] := 3.6455727, [22] := 3.6455727, [23] := 3.6455727, [24] := 3.6455727, [25] := 3.6455727, [26] := 3.6455727, [27] := 3.6455727, [28] := 3.6455727, [29] := 3.6455727, [30] := 3.6455727, [31] := 3.6455727, [32] := 3.6455727, [33] := 3.6455727, [34] := 3.6455727, [35] := 3.6455727, [36] := 3.6455727, [37] := 3.6455727, [38] := 3.6455727, [39] := 3.6455727, [40] := 3.6455727, [41] := 3.6455727, [42] := 3.6455727, [43] := 3.6455727, [44] := 3.6455727, [45] := 3.6455727, [46] := 3.6455727, [47] := 3.6455727, [48] := 3.6455727, [49] := 3.6455727, [50] := 3.6455727, [51] := 3.6455727, [52] := 3.6455727, [53] := 3.6455727, [54] := 3.6455727, [55] := 3.6455727, [56] := 3.6455727, [57] := 3.6455727, [58] := 3.6455727, [59] := 3.6455727);   // 650 length array with flow values for insp O2 valve, set by calcBreath()
   O2 : DINT;
   O2ConstantFlow : REAL := 3.6455727;
   O2Down : CAM_PROFILE[1010] := ([0].Status := 2, [1].Status := 2, [2].Status := 2, [3].Status := 2, [4].Status := 2, [5].Status := 2, [6].Status := 2, [7].Status := 2, [8].Status := 2, [9].Status := 2, [10].Status := 2, [11].Status := 2, [12].Status := 2, [13].Status := 2, [14].Status := 2, [15].Status := 2, [16].Status := 2, [17].Status := 2, [18].Status := 2, [19].Status := 2, [20].Status := 2, [21].Status := 2, [22].Status := 2, [23].Status := 2, [24].Status := 2, [25].Status := 2, [26].Status := 2, [27].Status := 2, [28].Status := 2, [29].Status := 2, [30].Status := 2, [31].Status := 2, [32].Status := 2, [33].Status := 2, [34].Status := 2, [35].Status := 2, [36].Status := 2, [37].Status := 2, [38].Status := 2, [39].Status := 2, [40].Status := 2, [41].Status := 2, [42].Status := 2, [43].Status := 2, [44].Status := 2, [45].Status := 2, [46].Status := 2, [47].Status := 2, [48].Status := 2, [49].Status := 2, [50].Status := 2, [51].Status := 2, [52].Status := 2, [53].Status := 2, [54].Status := 2, [55].Status := 2, [56].Status := 2, [57].Status := 2, [58].Status := 2, [59].Status := 2,
        [60].Status := 2, [61].Status := 2, [62].Status := 2, [63].Status := 2, [64].Status := 2, [65].Status := 2, [66].Status := 2, [67].Status := 2, [68].Status := 2, [69].Status := 2, [70].Status := 2, [71].Status := 2, [72].Status := 2, [73].Status := 2, [74].Status := 2, [75].Status := 2, [76].Status := 2, [77].Status := 2, [78].Status := 2, [79].Status := 2, [80].Status := 2, [81].Status := 2, [82].Status := 2, [83].Status := 2, [84].Status := 2, [85].Status := 2, [86].Status := 2, [87].Status := 2, [88].Status := 2, [89].Status := 2, [90].Status := 2, [91].Status := 2, [92].Status := 2, [93].Status := 2, [94].Status := 2, [95].Status := 2, [96].Status := 2, [97].Status := 2, [98].Status := 2, [99].Status := 2, [100].Status := 2, [101].Status := 2, [102].Status := 2, [103].Status := 2, [104].Status := 2, [105].Status := 2, [106].Status := 2, [107].Status := 2, [108].Status := 2, [109].Status := 2, [110].Status := 2, [111].Status := 2, [112].Status := 2, [113].Status := 2, [114].Status := 2, [115].Status := 2, [116].Status := 2, [117].Status := 2, [118].Status := 2, [119].Status := 2,
        [120].Status := 2, [121].Status := 2, [122].Status := 2, [123].Status := 2, [124].Status := 2, [125].Status := 2, [126].Status := 2, [127].Status := 2, [128].Status := 2, [129].Status := 2, [130].Status := 2, [131].Status := 2, [132].Status := 2, [133].Status := 2, [134].Status := 2, [135].Status := 2, [136].Status := 2, [137].Status := 2, [138].Status := 2, [139].Status := 2, [140].Status := 2, [141].Status := 2, [142].Status := 2, [143].Status := 2, [144].Status := 2, [145].Status := 2, [146].Status := 2, [147].Status := 2, [148].Status := 2, [149].Status := 2, [150].Status := 2, [151].Status := 2, [152].Status := 2, [153].Status := 2, [154].Status := 2, [155].Status := 2, [156].Status := 2, [157].Status := 2, [158].Status := 2, [159].Status := 2, [160].Status := 2, [161].Status := 2, [162].Status := 2, [163].Status := 2, [164].Status := 2, [165].Status := 2, [166].Status := 2, [167].Status := 2, [168].Status := 2, [169].Status := 2, [170].Status := 2, [171].Status := 2, [172].Status := 2, [173].Status := 2, [174].Status := 2, [175].Status := 2, [176].Status := 2, [177].Status := 2, [178].Status := 2, [179].Status := 2,
        [180].Status := 2, [181].Status := 2, [182].Status := 2, [183].Status := 2, [184].Status := 2, [185].Status := 2, [186].Status := 2, [187].Status := 2, [188].Status := 2, [189].Status := 2, [190].Status := 2, [191].Status := 2, [192].Status := 2, [193].Status := 2, [194].Status := 2, [195].Status := 2, [196].Status := 2, [197].Status := 2, [198].Status := 2, [199].Status := 2, [200].Status := 2, [201].Status := 2, [202].Status := 2, [203].Status := 2, [204].Status := 2, [205].Status := 2, [206].Status := 2, [207].Status := 2, [208].Status := 2, [209].Status := 2, [210].Status := 2, [211].Status := 2, [212].Status := 2, [213].Status := 2, [214].Status := 2, [215].Status := 2, [216].Status := 2, [217].Status := 2, [218].Status := 2, [219].Status := 2, [220].Status := 2, [221].Status := 2, [222].Status := 2, [223].Status := 2, [224].Status := 2, [225].Status := 2, [226].Status := 2, [227].Status := 2, [228].Status := 2, [229].Status := 2, [230].Status := 2, [231].Status := 2, [232].Status := 2, [233].Status := 2, [234].Status := 2, [235].Status := 2, [236].Status := 2, [237].Status := 2, [238].Status := 2, [239].Status := 2,
        [240].Status := 2, [241].Status := 2, [242].Status := 2, [243].Status := 2, [244].Status := 2, [245].Status := 2, [246].Status := 2, [247].Status := 2, [248].Status := 2, [249].Status := 2, [250].Status := 2, [251].Status := 2, [252].Status := 2, [253].Status := 2, [254].Status := 2, [255].Status := 2, [256].Status := 2, [257].Status := 2, [258].Status := 2, [259].Status := 2, [260].Status := 2, [261].Status := 2, [262].Status := 2, [263].Status := 2, [264].Status := 2, [265].Status := 2, [266].Status := 2, [267].Status := 2, [268].Status := 2, [269].Status := 2, [270].Status := 2, [271].Status := 2, [272].Status := 2, [273].Status := 2, [274].Status := 2, [275].Status := 2, [276].Status := 2, [277].Status := 2, [278].Status := 2, [279].Status := 2, [280].Status := 2, [281].Status := 2, [282].Status := 2, [283].Status := 2, [284].Status := 2, [285].Status := 2, [286].Status := 2, [287].Status := 2, [288].Status := 2, [289].Status := 2, [290].Status := 2, [291].Status := 2, [292].Status := 2, [293].Status := 2, [294].Status := 2, [295].Status := 2, [296].Status := 2, [297].Status := 2, [298].Status := 2, [299].Status := 2,
        [300].Status := 2, [301].Status := 2, [302].Status := 2, [303].Status := 2, [304].Status := 2, [305].Status := 2, [306].Status := 2, [307].Status := 2, [308].Status := 2, [309].Status := 2, [310].Status := 2, [311].Status := 2, [312].Status := 2, [313].Status := 2, [314].Status := 2, [315].Status := 2, [316].Status := 2, [317].Status := 2, [318].Status := 2, [319].Status := 2, [320].Status := 2, [321].Status := 2, [322].Status := 2, [323].Status := 2, [324].Status := 2, [325].Status := 2, [326].Status := 2, [327].Status := 2, [328].Status := 2, [329].Status := 2, [330].Status := 2, [331].Status := 2, [332].Status := 2, [333].Status := 2, [334].Status := 2, [335].Status := 2, [336].Status := 2, [337].Status := 2, [338].Status := 2, [339].Status := 2, [340].Status := 2, [341].Status := 2, [342].Status := 2, [343].Status := 2, [344].Status := 2, [345].Status := 2, [346].Status := 2, [347].Status := 2, [348].Status := 2, [349].Status := 2, [350].Status := 2, [351].Status := 2, [352].Status := 2, [353].Status := 2, [354].Status := 2, [355].Status := 2, [356].Status := 2, [357].Status := 2, [358].Status := 2, [359].Status := 2,
        [360].Status := 2, [361].Status := 2, [362].Status := 2, [363].Status := 2, [364].Status := 2, [365].Status := 2, [366].Status := 2, [367].Status := 2, [368].Status := 2, [369].Status := 2, [370].Status := 2, [371].Status := 2, [372].Status := 2, [373].Status := 2, [374].Status := 2, [375].Status := 2, [376].Status := 2, [377].Status := 2, [378].Status := 2, [379].Status := 2, [380].Status := 2, [381].Status := 2, [382].Status := 2, [383].Status := 2, [384].Status := 2, [385].Status := 2, [386].Status := 2, [387].Status := 2, [388].Status := 2, [389].Status := 2, [390].Status := 2, [391].Status := 2, [392].Status := 2, [393].Status := 2, [394].Status := 2, [395].Status := 2, [396].Status := 2, [397].Status := 2, [398].Status := 2, [399].Status := 2, [400].Status := 2, [401].Status := 2, [402].Status := 2, [403].Status := 2, [404].Status := 2, [405].Status := 2, [406].Status := 2, [407].Status := 2, [408].Status := 2, [409].Status := 2, [410].Status := 2, [411].Status := 2, [412].Status := 2, [413].Status := 2, [414].Status := 2, [415].Status := 2, [416].Status := 2, [417].Status := 2, [418].Status := 2, [419].Status := 2,
        [420].Status := 2, [421].Status := 2, [422].Status := 2, [423].Status := 2, [424].Status := 2, [425].Status := 2, [426].Status := 2, [427].Status := 2, [428].Status := 2, [429].Status := 2, [430].Status := 2, [431].Status := 2, [432].Status := 2, [433].Status := 2, [434].Status := 2, [435].Status := 2, [436].Status := 2, [437].Status := 2, [438].Status := 2, [439].Status := 2, [440].Status := 2, [441].Status := 2, [442].Status := 2, [443].Status := 2, [444].Status := 2, [445].Status := 2, [446].Status := 2, [447].Status := 2, [448].Status := 2, [449].Status := 2, [450].Status := 2, [451].Status := 2, [452].Status := 2, [453].Status := 2, [454].Status := 2, [455].Status := 2, [456].Status := 2, [457].Status := 2, [458].Status := 2, [459].Status := 2, [460].Status := 2, [461].Status := 2, [462].Status := 2, [463].Status := 2, [464].Status := 2, [465].Status := 2, [466].Status := 2, [467].Status := 2, [468].Status := 2, [469].Status := 2, [470].Status := 2, [471].Status := 2, [472].Status := 2, [473].Status := 2, [474].Status := 2, [475].Status := 2, [476].Status := 2, [477].Status := 2, [478].Status := 2, [479].Status := 2,
        [480].Status := 2, [481].Status := 2, [482].Status := 2, [483].Status := 2, [484].Status := 2, [485].Status := 2, [486].Status := 2, [487].Status := 2, [488].Status := 2, [489].Status := 2, [490].Status := 2, [491].Status := 2, [492].Status := 2, [493].Status := 2, [494].Status := 2, [495].Status := 2, [496].Status := 2, [497].Status := 2, [498].Status := 2, [499].Status := 2, [500].Status := 2, [501].Status := 2, [502].Status := 2, [503].Status := 2, [504].Status := 2, [505].Status := 2, [506].Status := 2, [507].Status := 2, [508].Status := 2, [509].Status := 2, [510].Status := 2, [511].Status := 2, [512].Status := 2, [513].Status := 2, [514].Status := 2, [515].Status := 2, [516].Status := 2, [517].Status := 2, [518].Status := 2, [519].Status := 2, [520].Status := 2, [521].Status := 2, [522].Status := 2, [523].Status := 2, [524].Status := 2, [525].Status := 2, [526].Status := 2, [527].Status := 2, [528].Status := 2, [529].Status := 2, [530].Status := 2, [531].Status := 2, [532].Status := 2, [533].Status := 2, [534].Status := 2, [535].Status := 2, [536].Status := 2, [537].Status := 2, [538].Status := 2, [539].Status := 2,
        [540].Status := 2, [541].Status := 2, [542].Status := 2, [543].Status := 2, [544].Status := 2, [545].Status := 2, [546].Status := 2, [547].Status := 2, [548].Status := 2, [549].Status := 2, [550].Status := 2, [551].Status := 2, [552].Status := 2, [553].Status := 2, [554].Status := 2, [555].Status := 2, [556].Status := 2, [557].Status := 2, [558].Status := 2, [559].Status := 2, [560].Status := 2, [561].Status := 2, [562].Status := 2, [563].Status := 2, [564].Status := 2, [565].Status := 2, [566].Status := 2, [567].Status := 2, [568].Status := 2, [569].Status := 2, [570].Status := 2, [571].Status := 2, [572].Status := 2, [573].Status := 2, [574].Status := 2, [575].Status := 2, [576].Status := 2, [577].Status := 2, [578].Status := 2, [579].Status := 2, [580].Status := 2, [581].Status := 2, [582].Status := 2, [583].Status := 2, [584].Status := 2, [585].Status := 2, [586].Status := 2, [587].Status := 2, [588].Status := 2, [589].Status := 2, [590].Status := 2, [591].Status := 2, [592].Status := 2, [593].Status := 2, [594].Status := 2, [595].Status := 2, [596].Status := 2, [597].Status := 2, [598].Status := 2, [599].Status := 2,
        [600].Status := 2, [601].Status := 2, [602].Status := 2, [603].Status := 2, [604].Status := 2, [605].Status := 2, [606].Status := 2, [607].Status := 2, [608].Status := 2, [609].Status := 2, [610].Status := 2, [611].Status := 2, [612].Status := 2, [613].Status := 2, [614].Status := 2, [615].Status := 2, [616].Status := 2, [617].Status := 2, [618].Status := 2, [619].Status := 2, [620].Status := 2, [621].Status := 2, [622].Status := 2, [623].Status := 2, [624].Status := 2, [625].Status := 2, [626].Status := 2, [627].Status := 2, [628].Status := 2, [629].Status := 2, [630].Status := 2, [631].Status := 2, [632].Status := 2, [633].Status := 2, [634].Status := 2, [635].Status := 2, [636].Status := 2, [637].Status := 2, [638].Status := 2, [639].Status := 2, [640].Status := 2, [641].Status := 2, [642].Status := 2, [643].Status := 2, [644].Status := 2, [645].Status := 2, [646].Status := 2, [647].Status := 2, [648].Status := 2, [649].Status := 2, [650].Status := 2, [651].Status := 2, [652].Status := 2, [653].Status := 2, [654].Status := 2, [655].Status := 2, [656].Status := 2, [657].Status := 2, [658].Status := 2, [659].Status := 2,
        [660].Status := 2, [661].Status := 2, [662].Status := 2, [663].Status := 2, [664].Status := 2, [665].Status := 2, [666].Status := 2, [667].Status := 2, [668].Status := 2, [669].Status := 2, [670].Status := 2, [671].Status := 2, [672].Status := 2, [673].Status := 2, [674].Status := 2, [675].Status := 2, [676].Status := 2, [677].Status := 2, [678].Status := 2, [679].Status := 2, [680].Status := 2, [681].Status := 2, [682].Status := 2, [683].Status := 2, [684].Status := 2, [685].Status := 2, [686].Status := 2, [687].Status := 2, [688].Status := 2, [689].Status := 2, [690].Status := 2, [691].Status := 2, [692].Status := 2, [693].Status := 2, [694].Status := 2, [695].Status := 2, [696].Status := 2, [697].Status := 2, [698].Status := 2, [699].Status := 2, [700].Status := 2, [701].Status := 2, [702].Status := 2, [703].Status := 2, [704].Status := 2, [705].Status := 2, [706].Status := 2, [707].Status := 2, [708].Status := 2, [709].Status := 2, [710].Status := 2, [711].Status := 2, [712].Status := 2, [713].Status := 2, [714].Status := 2, [715].Status := 2, [716].Status := 2, [717].Status := 2, [718].Status := 2, [719].Status := 2,
        [720].Status := 2, [721].Status := 2, [722].Status := 2, [723].Status := 2, [724].Status := 2, [725].Status := 2, [726].Status := 2, [727].Status := 2, [728].Status := 2, [729].Status := 2, [730].Status := 2, [731].Status := 2, [732].Status := 2, [733].Status := 2, [734].Status := 2, [735].Status := 2, [736].Status := 2, [737].Status := 2, [738].Status := 2, [739].Status := 2, [740].Status := 2, [741].Status := 2, [742].Status := 2, [743].Status := 2, [744].Status := 2, [745].Status := 2, [746].Status := 2, [747].Status := 2, [748].Status := 2, [749].Status := 2, [750].Status := 2, [751].Status := 2, [752].Status := 2, [753].Status := 2, [754].Status := 2, [755].Status := 2, [756].Status := 2, [757].Status := 2, [758].Status := 2, [759].Status := 2, [760].Status := 2, [761].Status := 2, [762].Status := 2, [763].Status := 2, [764].Status := 2, [765].Status := 2, [766].Status := 2, [767].Status := 2, [768].Status := 2, [769].Status := 2, [770].Status := 2, [771].Status := 2, [772].Status := 2, [773].Status := 2, [774].Status := 2, [775].Status := 2, [776].Status := 2, [777].Status := 2, [778].Status := 2, [779].Status := 2,
        [780].Status := 2, [781].Status := 2, [782].Status := 2, [783].Status := 2, [784].Status := 2, [785].Status := 2, [786].Status := 2, [787].Status := 2, [788].Status := 2, [789].Status := 2, [790].Status := 2, [791].Status := 2, [792].Status := 2, [793].Status := 2, [794].Status := 2, [795].Status := 2, [796].Status := 2, [797].Status := 2, [798].Status := 2, [799].Status := 2, [800].Status := 2, [801].Status := 2, [802].Status := 2, [803].Status := 2, [804].Status := 2, [805].Status := 2, [806].Status := 2, [807].Status := 2, [808].Status := 2, [809].Status := 2, [810].Status := 2, [811].Status := 2, [812].Status := 2, [813].Status := 2, [814].Status := 2, [815].Status := 2, [816].Status := 2, [817].Status := 2, [818].Status := 2, [819].Status := 2, [820].Status := 2, [821].Status := 2, [822].Status := 2, [823].Status := 2, [824].Status := 2, [825].Status := 2, [826].Status := 2, [827].Status := 2, [828].Status := 2, [829].Status := 2, [830].Status := 2, [831].Status := 2, [832].Status := 2, [833].Status := 2, [834].Status := 2, [835].Status := 2, [836].Status := 2, [837].Status := 2, [838].Status := 2, [839].Status := 2,
        [840].Status := 2, [841].Status := 2, [842].Status := 2, [843].Status := 2, [844].Status := 2, [845].Status := 2, [846].Status := 2, [847].Status := 2, [848].Status := 2, [849].Status := 2, [850].Status := 2, [851].Status := 2, [852].Status := 2, [853].Status := 2, [854].Status := 2, [855].Status := 2, [856].Status := 2, [857].Status := 2, [858].Status := 2, [859].Status := 2, [860].Status := 2, [861].Status := 2, [862].Status := 2, [863].Status := 2, [864].Status := 2, [865].Status := 2, [866].Status := 2, [867].Status := 2, [868].Status := 2, [869].Status := 2, [870].Status := 2, [871].Status := 2, [872].Status := 2, [873].Status := 2, [874].Status := 2, [875].Status := 2, [876].Status := 2, [877].Status := 2, [878].Status := 2, [879].Status := 2, [880].Status := 2, [881].Status := 2, [882].Status := 2, [883].Status := 2, [884].Status := 2, [885].Status := 2, [886].Status := 2, [887].Status := 2, [888].Status := 2, [889].Status := 2, [890].Status := 2, [891].Status := 2, [892].Status := 2, [893].Status := 2, [894].Status := 2, [895].Status := 2, [896].Status := 2, [897].Status := 2, [898].Status := 2, [899].Status := 2,
        [900].Status := 2, [901].Status := 2, [902].Status := 2, [903].Status := 2, [904].Status := 2, [905].Status := 2, [906].Status := 2, [907].Status := 2, [908].Status := 2, [909].Status := 2, [910].Status := 2, [911].Status := 2, [912].Status := 2, [913].Status := 2, [914].Status := 2, [915].Status := 2, [916].Status := 2, [917].Status := 2, [918].Status := 2, [919].Status := 2, [920].Status := 2, [921].Status := 2, [922].Status := 2, [923].Status := 2, [924].Status := 2, [925].Status := 2, [926].Status := 2, [927].Status := 2, [928].Status := 2, [929].Status := 2, [930].Status := 2, [931].Status := 2, [932].Status := 2, [933].Status := 2, [934].Status := 2, [935].Status := 2, [936].Status := 2, [937].Status := 2, [938].Status := 2, [939].Status := 2, [940].Status := 2, [941].Status := 2, [942].Status := 2, [943].Status := 2, [944].Status := 2, [945].Status := 2, [946].Status := 2, [947].Status := 2, [948].Status := 2, [949].Status := 2, [950].Status := 2, [951].Status := 2, [952].Status := 2, [953].Status := 2, [954].Status := 2, [955].Status := 2, [956].Status := 2, [957].Status := 2, [958].Status := 2, [959].Status := 2,
        [960].Status := 2, [961].Status := 2, [962].Status := 2, [963].Status := 2, [964].Status := 2, [965].Status := 2, [966].Status := 2, [967].Status := 2, [968].Status := 2, [969].Status := 2, [970].Status := 2, [971].Status := 2, [972].Status := 2, [973].Status := 2, [974].Status := 2, [975].Status := 2, [976].Status := 2, [977].Status := 2, [978].Status := 2, [979].Status := 2, [980].Status := 2, [981].Status := 2, [982].Status := 2, [983].Status := 2, [984].Status := 2, [985].Status := 2, [986].Status := 2, [987].Status := 2, [988].Status := 2, [989].Status := 2, [990].Status := 2, [991].Status := 2, [992].Status := 2, [993].Status := 2, [994].Status := 2, [995].Status := 2, [996].Status := 2, [997].Status := 2, [998].Status := 2, [999].Status := 2, [1000].Status := 2, [1001].Status := 2, [1002].Status := 2);
   O2mADer : REAL;
   O2mAOut : REAL;
   O2mASlope : REAL := 416748.25;
   O2RampFlowIncreasePerAdjust : REAL := 0.18227863;
   O2Up : CAM_PROFILE[1010] := ([0].Status := 2, [1].Status := 2, [2].Status := 2, [3].Status := 2, [4].Status := 2, [5].Status := 2, [6].Status := 2, [7].Status := 2, [8].Status := 2, [9].Status := 2, [10].Status := 2, [11].Status := 2, [12].Status := 2, [13].Status := 2, [14].Status := 2, [15].Status := 2, [16].Status := 2, [17].Status := 2, [18].Status := 2, [19].Status := 2, [20].Status := 2, [21].Status := 2, [22].Status := 2, [23].Status := 2, [24].Status := 2, [25].Status := 2, [26].Status := 2, [27].Status := 2, [28].Status := 2, [29].Status := 2, [30].Status := 2, [31].Status := 2, [32].Status := 2, [33].Status := 2, [34].Status := 2, [35].Status := 2, [36].Status := 2, [37].Status := 2, [38].Status := 2, [39].Status := 2, [40].Status := 2, [41].Status := 2, [42].Status := 2, [43].Status := 2, [44].Status := 2, [45].Status := 2, [46].Status := 2, [47].Status := 2, [48].Status := 2, [49].Status := 2, [50].Status := 2, [51].Status := 2, [52].Status := 2, [53].Status := 2, [54].Status := 2, [55].Status := 2, [56].Status := 2, [57].Status := 2, [58].Status := 2, [59].Status := 2,
        [60].Status := 2, [61].Status := 2, [62].Status := 2, [63].Status := 2, [64].Status := 2, [65].Status := 2, [66].Status := 2, [67].Status := 2, [68].Status := 2, [69].Status := 2, [70].Status := 2, [71].Status := 2, [72].Status := 2, [73].Status := 2, [74].Status := 2, [75].Status := 2, [76].Status := 2, [77].Status := 2, [78].Status := 2, [79].Status := 2, [80].Status := 2, [81].Status := 2, [82].Status := 2, [83].Status := 2, [84].Status := 2, [85].Status := 2, [86].Status := 2, [87].Status := 2, [88].Status := 2, [89].Status := 2, [90].Status := 2, [91].Status := 2, [92].Status := 2, [93].Status := 2, [94].Status := 2, [95].Status := 2, [96].Status := 2, [97].Status := 2, [98].Status := 2, [99].Status := 2, [100].Status := 2, [101].Status := 2, [102].Status := 2, [103].Status := 2, [104].Status := 2, [105].Status := 2, [106].Status := 2, [107].Status := 2, [108].Status := 2, [109].Status := 2, [110].Status := 2, [111].Status := 2, [112].Status := 2, [113].Status := 2, [114].Status := 2, [115].Status := 2, [116].Status := 2, [117].Status := 2, [118].Status := 2, [119].Status := 2,
        [120].Status := 2, [121].Status := 2, [122].Status := 2, [123].Status := 2, [124].Status := 2, [125].Status := 2, [126].Status := 2, [127].Status := 2, [128].Status := 2, [129].Status := 2, [130].Status := 2, [131].Status := 2, [132].Status := 2, [133].Status := 2, [134].Status := 2, [135].Status := 2, [136].Status := 2, [137].Status := 2, [138].Status := 2, [139].Status := 2, [140].Status := 2, [141].Status := 2, [142].Status := 2, [143].Status := 2, [144].Status := 2, [145].Status := 2, [146].Status := 2, [147].Status := 2, [148].Status := 2, [149].Status := 2, [150].Status := 2, [151].Status := 2, [152].Status := 2, [153].Status := 2, [154].Status := 2, [155].Status := 2, [156].Status := 2, [157].Status := 2, [158].Status := 2, [159].Status := 2, [160].Status := 2, [161].Status := 2, [162].Status := 2, [163].Status := 2, [164].Status := 2, [165].Status := 2, [166].Status := 2, [167].Status := 2, [168].Status := 2, [169].Status := 2, [170].Status := 2, [171].Status := 2, [172].Status := 2, [173].Status := 2, [174].Status := 2, [175].Status := 2, [176].Status := 2, [177].Status := 2, [178].Status := 2, [179].Status := 2,
        [180].Status := 2, [181].Status := 2, [182].Status := 2, [183].Status := 2, [184].Status := 2, [185].Status := 2, [186].Status := 2, [187].Status := 2, [188].Status := 2, [189].Status := 2, [190].Status := 2, [191].Status := 2, [192].Status := 2, [193].Status := 2, [194].Status := 2, [195].Status := 2, [196].Status := 2, [197].Status := 2, [198].Status := 2, [199].Status := 2, [200].Status := 2, [201].Status := 2, [202].Status := 2, [203].Status := 2, [204].Status := 2, [205].Status := 2, [206].Status := 2, [207].Status := 2, [208].Status := 2, [209].Status := 2, [210].Status := 2, [211].Status := 2, [212].Status := 2, [213].Status := 2, [214].Status := 2, [215].Status := 2, [216].Status := 2, [217].Status := 2, [218].Status := 2, [219].Status := 2, [220].Status := 2, [221].Status := 2, [222].Status := 2, [223].Status := 2, [224].Status := 2, [225].Status := 2, [226].Status := 2, [227].Status := 2, [228].Status := 2, [229].Status := 2, [230].Status := 2, [231].Status := 2, [232].Status := 2, [233].Status := 2, [234].Status := 2, [235].Status := 2, [236].Status := 2, [237].Status := 2, [238].Status := 2, [239].Status := 2,
        [240].Status := 2, [241].Status := 2, [242].Status := 2, [243].Status := 2, [244].Status := 2, [245].Status := 2, [246].Status := 2, [247].Status := 2, [248].Status := 2, [249].Status := 2, [250].Status := 2, [251].Status := 2, [252].Status := 2, [253].Status := 2, [254].Status := 2, [255].Status := 2, [256].Status := 2, [257].Status := 2, [258].Status := 2, [259].Status := 2, [260].Status := 2, [261].Status := 2, [262].Status := 2, [263].Status := 2, [264].Status := 2, [265].Status := 2, [266].Status := 2, [267].Status := 2, [268].Status := 2, [269].Status := 2, [270].Status := 2, [271].Status := 2, [272].Status := 2, [273].Status := 2, [274].Status := 2, [275].Status := 2, [276].Status := 2, [277].Status := 2, [278].Status := 2, [279].Status := 2, [280].Status := 2, [281].Status := 2, [282].Status := 2, [283].Status := 2, [284].Status := 2, [285].Status := 2, [286].Status := 2, [287].Status := 2, [288].Status := 2, [289].Status := 2, [290].Status := 2, [291].Status := 2, [292].Status := 2, [293].Status := 2, [294].Status := 2, [295].Status := 2, [296].Status := 2, [297].Status := 2, [298].Status := 2, [299].Status := 2,
        [300].Status := 2, [301].Status := 2, [302].Status := 2, [303].Status := 2, [304].Status := 2, [305].Status := 2, [306].Status := 2, [307].Status := 2, [308].Status := 2, [309].Status := 2, [310].Status := 2, [311].Status := 2, [312].Status := 2, [313].Status := 2, [314].Status := 2, [315].Status := 2, [316].Status := 2, [317].Status := 2, [318].Status := 2, [319].Status := 2, [320].Status := 2, [321].Status := 2, [322].Status := 2, [323].Status := 2, [324].Status := 2, [325].Status := 2, [326].Status := 2, [327].Status := 2, [328].Status := 2, [329].Status := 2, [330].Status := 2, [331].Status := 2, [332].Status := 2, [333].Status := 2, [334].Status := 2, [335].Status := 2, [336].Status := 2, [337].Status := 2, [338].Status := 2, [339].Status := 2, [340].Status := 2, [341].Status := 2, [342].Status := 2, [343].Status := 2, [344].Status := 2, [345].Status := 2, [346].Status := 2, [347].Status := 2, [348].Status := 2, [349].Status := 2, [350].Status := 2, [351].Status := 2, [352].Status := 2, [353].Status := 2, [354].Status := 2, [355].Status := 2, [356].Status := 2, [357].Status := 2, [358].Status := 2, [359].Status := 2,
        [360].Status := 2, [361].Status := 2, [362].Status := 2, [363].Status := 2, [364].Status := 2, [365].Status := 2, [366].Status := 2, [367].Status := 2, [368].Status := 2, [369].Status := 2, [370].Status := 2, [371].Status := 2, [372].Status := 2, [373].Status := 2, [374].Status := 2, [375].Status := 2, [376].Status := 2, [377].Status := 2, [378].Status := 2, [379].Status := 2, [380].Status := 2, [381].Status := 2, [382].Status := 2, [383].Status := 2, [384].Status := 2, [385].Status := 2, [386].Status := 2, [387].Status := 2, [388].Status := 2, [389].Status := 2, [390].Status := 2, [391].Status := 2, [392].Status := 2, [393].Status := 2, [394].Status := 2, [395].Status := 2, [396].Status := 2, [397].Status := 2, [398].Status := 2, [399].Status := 2, [400].Status := 2, [401].Status := 2, [402].Status := 2, [403].Status := 2, [404].Status := 2, [405].Status := 2, [406].Status := 2, [407].Status := 2, [408].Status := 2, [409].Status := 2, [410].Status := 2, [411].Status := 2, [412].Status := 2, [413].Status := 2, [414].Status := 2, [415].Status := 2, [416].Status := 2, [417].Status := 2, [418].Status := 2, [419].Status := 2,
        [420].Status := 2, [421].Status := 2, [422].Status := 2, [423].Status := 2, [424].Status := 2, [425].Status := 2, [426].Status := 2, [427].Status := 2, [428].Status := 2, [429].Status := 2, [430].Status := 2, [431].Status := 2, [432].Status := 2, [433].Status := 2, [434].Status := 2, [435].Status := 2, [436].Status := 2, [437].Status := 2, [438].Status := 2, [439].Status := 2, [440].Status := 2, [441].Status := 2, [442].Status := 2, [443].Status := 2, [444].Status := 2, [445].Status := 2, [446].Status := 2, [447].Status := 2, [448].Status := 2, [449].Status := 2, [450].Status := 2, [451].Status := 2, [452].Status := 2, [453].Status := 2, [454].Status := 2, [455].Status := 2, [456].Status := 2, [457].Status := 2, [458].Status := 2, [459].Status := 2, [460].Status := 2, [461].Status := 2, [462].Status := 2, [463].Status := 2, [464].Status := 2, [465].Status := 2, [466].Status := 2, [467].Status := 2, [468].Status := 2, [469].Status := 2, [470].Status := 2, [471].Status := 2, [472].Status := 2, [473].Status := 2, [474].Status := 2, [475].Status := 2, [476].Status := 2, [477].Status := 2, [478].Status := 2, [479].Status := 2,
        [480].Status := 2, [481].Status := 2, [482].Status := 2, [483].Status := 2, [484].Status := 2, [485].Status := 2, [486].Status := 2, [487].Status := 2, [488].Status := 2, [489].Status := 2, [490].Status := 2, [491].Status := 2, [492].Status := 2, [493].Status := 2, [494].Status := 2, [495].Status := 2, [496].Status := 2, [497].Status := 2, [498].Status := 2, [499].Status := 2, [500].Status := 2, [501].Status := 2, [502].Status := 2, [503].Status := 2, [504].Status := 2, [505].Status := 2, [506].Status := 2, [507].Status := 2, [508].Status := 2, [509].Status := 2, [510].Status := 2, [511].Status := 2, [512].Status := 2, [513].Status := 2, [514].Status := 2, [515].Status := 2, [516].Status := 2, [517].Status := 2, [518].Status := 2, [519].Status := 2, [520].Status := 2, [521].Status := 2, [522].Status := 2, [523].Status := 2, [524].Status := 2, [525].Status := 2, [526].Status := 2, [527].Status := 2, [528].Status := 2, [529].Status := 2, [530].Status := 2, [531].Status := 2, [532].Status := 2, [533].Status := 2, [534].Status := 2, [535].Status := 2, [536].Status := 2, [537].Status := 2, [538].Status := 2, [539].Status := 2,
